(* CoDeSys 2.3.9.48 project: 20171120_WUR.pro *)
(* Version: 0.9 *)
(* Description: Project Distributie Automatisering *)
(* Libraries: Serial_Interface_01.lib 22.4.13 11:50:14, Util.lib 30.1.13 12:05:12, WagoLib787_01.lib 10.11.14 12:02:32, mod_com.lib 30.1.13 12:05:12, WagoConfigToolLIB.lib 30.1.13 12:05:12, PowerMeasurement_495_02.lib 25.8.17 14:41:17, SysLibTime.lib 30.1.13 12:05:12, WagoLibSHA1.lib 19.8.11 13:53:16, WagoLibMySQL_03.lib 23.7.14 08:13:36, SerComm.lib 30.1.13 12:05:12, SysLibSockets.lib 22.5.14 15:16:32, SysLibFile.lib 30.1.13 12:05:12, SysLibMem.lib 30.1.13 12:05:12, SysLibSem.lib 30.1.13 12:05:12, SysLibRtc.lib 30.1.13 12:05:12, WagoLibEthernet_01.lib 1.4.15 13:24:28, WAGOLIBNTP.lib 19.8.11 13:53:14, Modb_l05.lib 13.5.15 09:30:08, SysLibDir.lib 30.1.13 12:05:12, Standard.lib 20.5.14 07:13:26, Iecsfc.lib 30.1.13 12:05:12, SYSLIBCALLBACK.LIB 30.1.13 12:05:12, WagoLibModbus_IP_01.lib 12.2.16 10:20:24, Wago_MBCFG_ETHERNET_01.lib 1.4.15 13:24:28, Wago_MBCFG_COMMON_01.lib 1.4.15 13:24:28 *)

(* PLC configuration (modules and I/O channels)
0750-0430 8 DI 24 V DC 3.0ms [Type_1_8_Channels] node 1, in %IB264 out %QB280
  AT %IX132.0 [BOOLOnX_I] Ch_1 Digital input
  AT %IX132.1 [BOOLOnX_I] Ch_2 Digital input
  AT %IX132.2 [BOOLOnX_I] Ch_3 Digital input
  AT %IX132.3 [BOOLOnX_I] Ch_4 Digital input
  AT %IX132.4 [BOOLOnX_I] Ch_5 Digital input
  AT %IX132.5 [BOOLOnX_I] Ch_6 Digital input
  AT %IX132.6 [BOOLOnX_I] Ch_7 Digital input
  AT %IX132.7 [BOOLOnX_I] Ch_8 Digital input
0750-0430 8 DI 24 V DC 3.0ms [Type_1_8_Channels] node 2, in %IB264 out %QB280
  AT %IX132.8 [BOOLOnX_I] Ch_1 Digital input
  AT %IX132.9 [BOOLOnX_I] Ch_2 Digital input
  AT %IX132.10 [BOOLOnX_I] Ch_3 Digital input
  AT %IX132.11 [BOOLOnX_I] Ch_4 Digital input
  AT %IX132.12 [BOOLOnX_I] Ch_5 Digital input
  AT %IX132.13 [BOOLOnX_I] Ch_6 Digital input
  AT %IX132.14 [BOOLOnX_I] Ch_7 Digital input
  AT %IX132.15 [BOOLOnX_I] Ch_8 Digital input
0750-0430 8 DI 24 V DC 3.0ms [Type_1_8_Channels] node 3, in %IB265 out %QB280
  AT %IX133.0 [BOOLOnX_I] Ch_1 Digital input
  AT %IX133.1 [BOOLOnX_I] Ch_2 Digital input
  AT %IX133.2 [BOOLOnX_I] Ch_3 Digital input
  AT %IX133.3 [BOOLOnX_I] Ch_4 Digital input
  AT %IX133.4 [BOOLOnX_I] Ch_5 Digital input
  AT %IX133.5 [BOOLOnX_I] Ch_6 Digital input
  AT %IX133.6 [BOOLOnX_I] Ch_7 Digital input
  AT %IX133.7 [BOOLOnX_I] Ch_8 Digital input
0750-0430 8 DI 24 V DC 3.0ms [Type_1_8_Channels] node 4, in %IB266 out %QB280
  AT %IX133.8 [BOOLOnX_I] Ch_1 Digital input
  AT %IX133.9 [BOOLOnX_I] Ch_2 Digital input
  AT %IX133.10 [BOOLOnX_I] Ch_3 Digital input
  AT %IX133.11 [BOOLOnX_I] Ch_4 Digital input
  AT %IX133.12 [BOOLOnX_I] Ch_5 Digital input
  AT %IX133.13 [BOOLOnX_I] Ch_6 Digital input
  AT %IX133.14 [BOOLOnX_I] Ch_7 Digital input
  AT %IX133.15 [BOOLOnX_I] Ch_8 Digital input
0750-0430 8 DI 24 V DC 3.0ms [Type_1_8_Channels] node 5, in %IB267 out %QB280
  AT %IX134.0 [BOOLOnX_I] Ch_1 Digital input
  AT %IX134.1 [BOOLOnX_I] Ch_2 Digital input
  AT %IX134.2 [BOOLOnX_I] Ch_3 Digital input
  AT %IX134.3 [BOOLOnX_I] Ch_4 Digital input
  AT %IX134.4 [BOOLOnX_I] Ch_5 Digital input
  AT %IX134.5 [BOOLOnX_I] Ch_6 Digital input
  AT %IX134.6 [BOOLOnX_I] Ch_7 Digital input
  AT %IX134.7 [BOOLOnX_I] Ch_8 Digital input
0750-0530 8 DO 24 V DC 0.5A [Type_10_8_Channels] node 6, in %IB268 out %QB280
  AT %QX140.0 [BOOLOnX_Q] Ch_1 Digital output
  AT %QX140.1 [BOOLOnX_Q] Ch_2 Digital output
  AT %QX140.2 [BOOLOnX_Q] Ch_3 Digital output
  AT %QX140.3 [BOOLOnX_Q] Ch_4 Digital output
  AT %QX140.4 [BOOLOnX_Q] Ch_5 Digital output
  AT %QX140.5 [BOOLOnX_Q] Ch_6 Digital output
  AT %QX140.6 [BOOLOnX_Q] Ch_7 Digital output
  AT %QX140.7 [BOOLOnX_Q] Ch_8 Digital output
0750-0530 8 DO 24 V DC 0.5A [Type_10_8_Channels] node 7, in %IB269 out %QB280
  AT %QX140.8 [BOOLOnX_Q] Ch_1 Digital output
  AT %QX140.9 [BOOLOnX_Q] Ch_2 Digital output
  AT %QX140.10 [BOOLOnX_Q] Ch_3 Digital output
  AT %QX140.11 [BOOLOnX_Q] Ch_4 Digital output
  AT %QX140.12 [BOOLOnX_Q] Ch_5 Digital output
  AT %QX140.13 [BOOLOnX_Q] Ch_6 Digital output
  AT %QX140.14 [BOOLOnX_Q] Ch_7 Digital output
  AT %QX140.15 [BOOLOnX_Q] Ch_8 Digital output
0750-0530 8 DO 24 V DC 0.5A [Type_10_8_Channels] node 8, in %IB269 out %QB281
  AT %QX141.0 [BOOLOnX_Q] Ch_1 Digital output
  AT %QX141.1 [BOOLOnX_Q] Ch_2 Digital output
  AT %QX141.2 [BOOLOnX_Q] Ch_3 Digital output
  AT %QX141.3 [BOOLOnX_Q] Ch_4 Digital output
  AT %QX141.4 [BOOLOnX_Q] Ch_5 Digital output
  AT %QX141.5 [BOOLOnX_Q] Ch_6 Digital output
  AT %QX141.6 [BOOLOnX_Q] Ch_7 Digital output
  AT %QX141.7 [BOOLOnX_Q] Ch_8 Digital output
0750-0530 8 DO 24 V DC 0.5A [Type_10_8_Channels] node 9, in %IB269 out %QB282
  AT %QX141.8 [BOOLOnX_Q] Ch_1 Digital output
  AT %QX141.9 [BOOLOnX_Q] Ch_2 Digital output
  AT %QX141.10 [BOOLOnX_Q] Ch_3 Digital output
  AT %QX141.11 [BOOLOnX_Q] Ch_4 Digital output
  AT %QX141.12 [BOOLOnX_Q] Ch_5 Digital output
  AT %QX141.13 [BOOLOnX_Q] Ch_6 Digital output
  AT %QX141.14 [BOOLOnX_Q] Ch_7 Digital output
  AT %QX141.15 [BOOLOnX_Q] Ch_8 Digital output
0750-0555 4 AO 4-20mA [Type_14_4_Channels] node 10, in %IB240 out %QB256
  AT %QW0 [WORDOnW_Q] Ch_1 Analog output
  AT %QW1 [WORDOnW_Q] Ch_2 Analog output
  AT %QW2 [WORDOnW_Q] Ch_3 Analog output
  AT %QW3 [WORDOnW_Q] Ch_4 Analog output
0750-0559 4 AO 0-10V DC [Type_14_4_Channels] node 11, in %IB240 out %QB256
  AT %QW4 [WORDOnW_Q] Ch_1 Analog output
  AT %QW5 [WORDOnW_Q] Ch_2 Analog output
  AT %QW6 [WORDOnW_Q] Ch_3 Analog output
  AT %QW7 [WORDOnW_Q] Ch_4 Analog output
0750-0495/0000-0001 3-phase PoM690/ 5A [Type_58_1_Channels] node 12, in %IB240 out %QB264
  AT %IW0 [WORDOnW_I] Status Word
  AT %IW1 [WORDOnW_I] Status Word 1
  AT %IW2 [WORDOnW_I] Status Word 2
  AT %IW3 [WORDOnW_I] Status Word 3
  AT %ID2 [DWORDOnD_I] process value 1
  AT %ID3 [DWORDOnD_I] process value 2
  AT %ID4 [DWORDOnD_I] process value 3
  AT %ID5 [DWORDOnD_I] process value 4
  AT %QW8 [WORDOnW_Q] Control Word
  AT %QW9 [WORDOnW_Q] Control Word 1
  AT %QW10 [WORDOnW_Q] Control Word 2
  AT %QW11 [WORDOnW_Q] Control Word 3
0750-0495/0000-0001 3-phase PoM690/ 5A [Type_58_1_Channels] node 13, in %IB240 out %QB272
  AT %IW12 [WORDOnW_I] Status Word
  AT %IW13 [WORDOnW_I] Status Word 1
  AT %IW14 [WORDOnW_I] Status Word 2
  AT %IW15 [WORDOnW_I] Status Word 3
  AT %ID8 [DWORDOnD_I] process value 1
  AT %ID9 [DWORDOnD_I] process value 2
  AT %ID10 [DWORDOnD_I] process value 3
  AT %ID11 [DWORDOnD_I] process value 4
  AT %QW20 [WORDOnW_Q] Control Word
  AT %QW21 [WORDOnW_Q] Control Word 1
  AT %QW22 [WORDOnW_Q] Control Word 2
  AT %QW23 [WORDOnW_Q] Control Word 3
0750-0495/0000-0001 3-phase PoM690/ 5A [Type_58_1_Channels] node 14, in %IB264 out %QB296
  AT %IW24 [WORDOnW_I] Status Word
  AT %IW25 [WORDOnW_I] Status Word 1
  AT %IW26 [WORDOnW_I] Status Word 2
  AT %IW27 [WORDOnW_I] Status Word 3
  AT %ID14 [DWORDOnD_I] process value 1
  AT %ID15 [DWORDOnD_I] process value 2
  AT %ID16 [DWORDOnD_I] process value 3
  AT %ID17 [DWORDOnD_I] process value 4
  AT %QW32 [WORDOnW_Q] Control Word
  AT %QW33 [WORDOnW_Q] Control Word 1
  AT %QW34 [WORDOnW_Q] Control Word 2
  AT %QW35 [WORDOnW_Q] Control Word 3
0750-0495/0000-0001 3-phase PoM690/ 5A [Type_58_1_Channels] node 15, in %IB288 out %QB320
  AT %IW36 [WORDOnW_I] Status Word
  AT %IW37 [WORDOnW_I] Status Word 1
  AT %IW38 [WORDOnW_I] Status Word 2
  AT %IW39 [WORDOnW_I] Status Word 3
  AT %ID20 [DWORDOnD_I] process value 1
  AT %ID21 [DWORDOnD_I] process value 2
  AT %ID22 [DWORDOnD_I] process value 3
  AT %ID23 [DWORDOnD_I] process value 4
  AT %QW44 [WORDOnW_Q] Control Word
  AT %QW45 [WORDOnW_Q] Control Word 1
  AT %QW46 [WORDOnW_Q] Control Word 2
  AT %QW47 [WORDOnW_Q] Control Word 3
0750-0495/0000-0001 3-phase PoM690/ 5A [Type_58_1_Channels] node 16, in %IB312 out %QB344
  AT %IW48 [WORDOnW_I] Status Word
  AT %IW49 [WORDOnW_I] Status Word 1
  AT %IW50 [WORDOnW_I] Status Word 2
  AT %IW51 [WORDOnW_I] Status Word 3
  AT %ID26 [DWORDOnD_I] process value 1
  AT %ID27 [DWORDOnD_I] process value 2
  AT %ID28 [DWORDOnD_I] process value 3
  AT %ID29 [DWORDOnD_I] process value 4
  AT %QW56 [WORDOnW_Q] Control Word
  AT %QW57 [WORDOnW_Q] Control Word 1
  AT %QW58 [WORDOnW_Q] Control Word 2
  AT %QW59 [WORDOnW_Q] Control Word 3
0750-0495/0000-0001 3-phase PoM690/ 5A [Type_58_1_Channels] node 17, in %IB336 out %QB368
  AT %IW60 [WORDOnW_I] Status Word
  AT %IW61 [WORDOnW_I] Status Word 1
  AT %IW62 [WORDOnW_I] Status Word 2
  AT %IW63 [WORDOnW_I] Status Word 3
  AT %ID32 [DWORDOnD_I] process value 1
  AT %ID33 [DWORDOnD_I] process value 2
  AT %ID34 [DWORDOnD_I] process value 3
  AT %ID35 [DWORDOnD_I] process value 4
  AT %QW68 [WORDOnW_Q] Control Word
  AT %QW69 [WORDOnW_Q] Control Word 1
  AT %QW70 [WORDOnW_Q] Control Word 2
  AT %QW71 [WORDOnW_Q] Control Word 3
0750-0495/0000-0001 3-phase PoM690/ 5A [Type_58_1_Channels] node 18, in %IB360 out %QB392
  AT %IW72 [WORDOnW_I] Status Word
  AT %IW73 [WORDOnW_I] Status Word 1
  AT %IW74 [WORDOnW_I] Status Word 2
  AT %IW75 [WORDOnW_I] Status Word 3
  AT %ID38 [DWORDOnD_I] process value 1
  AT %ID39 [DWORDOnD_I] process value 2
  AT %ID40 [DWORDOnD_I] process value 3
  AT %ID41 [DWORDOnD_I] process value 4
  AT %QW80 [WORDOnW_Q] Control Word
  AT %QW81 [WORDOnW_Q] Control Word 1
  AT %QW82 [WORDOnW_Q] Control Word 2
  AT %QW83 [WORDOnW_Q] Control Word 3
0750-0495/0000-0001 3-phase PoM690/ 5A [Type_58_1_Channels] node 19, in %IB384 out %QB416
  AT %IW84 [WORDOnW_I] Status Word
  AT %IW85 [WORDOnW_I] Status Word 1
  AT %IW86 [WORDOnW_I] Status Word 2
  AT %IW87 [WORDOnW_I] Status Word 3
  AT %ID44 [DWORDOnD_I] process value 1
  AT %ID45 [DWORDOnD_I] process value 2
  AT %ID46 [DWORDOnD_I] process value 3
  AT %ID47 [DWORDOnD_I] process value 4
  AT %QW92 [WORDOnW_Q] Control Word
  AT %QW93 [WORDOnW_Q] Control Word 1
  AT %QW94 [WORDOnW_Q] Control Word 2
  AT %QW95 [WORDOnW_Q] Control Word 3
0750-0495/0000-0001 3-phase PoM690/ 5A [Type_58_1_Channels] node 20, in %IB408 out %QB440
  AT %IW96 [WORDOnW_I] Status Word
  AT %IW97 [WORDOnW_I] Status Word 1
  AT %IW98 [WORDOnW_I] Status Word 2
  AT %IW99 [WORDOnW_I] Status Word 3
  AT %ID50 [DWORDOnD_I] process value 1
  AT %ID51 [DWORDOnD_I] process value 2
  AT %ID52 [DWORDOnD_I] process value 3
  AT %ID53 [DWORDOnD_I] process value 4
  AT %QW104 [WORDOnW_Q] Control Word
  AT %QW105 [WORDOnW_Q] Control Word 1
  AT %QW106 [WORDOnW_Q] Control Word 2
  AT %QW107 [WORDOnW_Q] Control Word 3
0750-0495/0000-0001 3-phase PoM690/ 5A [Type_58_1_Channels] node 21, in %IB432 out %QB464
  AT %IW108 [WORDOnW_I] Status Word
  AT %IW109 [WORDOnW_I] Status Word 1
  AT %IW110 [WORDOnW_I] Status Word 2
  AT %IW111 [WORDOnW_I] Status Word 3
  AT %ID56 [DWORDOnD_I] process value 1
  AT %ID57 [DWORDOnD_I] process value 2
  AT %ID58 [DWORDOnD_I] process value 3
  AT %ID59 [DWORDOnD_I] process value 4
  AT %QW116 [WORDOnW_Q] Control Word
  AT %QW117 [WORDOnW_Q] Control Word 1
  AT %QW118 [WORDOnW_Q] Control Word 2
  AT %QW119 [WORDOnW_Q] Control Word 3
0750-0495/0000-0001 3-phase PoM690/ 5A [Type_58_1_Channels] node 22, in %IB456 out %QB488
  AT %IW120 [WORDOnW_I] Status Word
  AT %IW121 [WORDOnW_I] Status Word 1
  AT %IW122 [WORDOnW_I] Status Word 2
  AT %IW123 [WORDOnW_I] Status Word 3
  AT %ID62 [DWORDOnD_I] process value 1
  AT %ID63 [DWORDOnD_I] process value 2
  AT %ID64 [DWORDOnD_I] process value 3
  AT %ID65 [DWORDOnD_I] process value 4
  AT %QW128 [WORDOnW_Q] Control Word
  AT %QW129 [WORDOnW_Q] Control Word 1
  AT %QW130 [WORDOnW_Q] Control Word 2
  AT %QW131 [WORDOnW_Q] Control Word 3
Modbus variables [PFC200MODBUS] node 1, in %IB0 out %QB0 {PlcStopBehaviour = 1; FiledbusErrorBehaviour = 1; TcpOperation = 1; TcpPort = 502; TcpTimeout = 600; UdpOperation = 1; UdpPort = 502; RtuOperation = 0; NodeId = 1; ResponseTimeout = 5000; Interface = 0; Baud = 115200; StopBits = 1; Parity = 1; FlowCtrl = 0; PhysInterface = 0}
  REAL, Fieldbus output [MODBUS_REAL_OUT] node 0, in %IB0 out %QB0
    mb_var0 AT %QD500 [REALOnD_Q] TEST
Modbus-Master [MB_MASTER] node 2, in %IB0 out %QB0
*)

(* Task configuration *)
TASK Test (PRIORITY := 2, INTERVAL := T#500ms);
	Group1();
END_TASK
TASK WriteData (PRIORITY := 29); (* freewheeling *)
	Main_logger();
	SystemStateNames();
END_TASK
TASK GroupSwitching (PRIORITY := 4, INTERVAL := T#1000ms);
	run_group_switching();
END_TASK
TASK TestCHPSwitch (PRIORITY := 25, INTERVAL := T#100ms);
	CHP_switch_delay();
END_TASK
TASK LightControl (PRIORITY := 31); (* freewheeling *)
	error_lights();
END_TASK
TASK Measurements (PRIORITY := 1, INTERVAL := T#200ms);
	run_PQ();
	variables_to_system_array();
END_TASK
TASK Control (PRIORITY := 5, INTERVAL := T#100ms);
	CHP_Controller();
	SOC_to_Voltage_Out();
	Mixer_Controller1();
	Mixer_Controller2();
END_TASK
TASK MB_ETH_MASTER_TASK (PRIORITY := 3, INTERVAL := T#100ms);
	MBCFG_Janitza_UMG5090();
END_TASK
TASK SyncSwitch (PRIORITY := 2, INTERVAL := T#50ms);
	run_synchroniser_swtich();
END_TASK

(* Global variable list: Global_Variables *)
VAR_GLOBAL
(* testing purpose values *)
	x																:	 REAL:=2;

(* internally used variables *)
	r_Battery_Bus_Frequency									:	 REAL;
	r_Battery_Bus_Voltage										:	 REAL;
	r_Grid_Bus_Frequency										:	 REAL;
	r_Grid_Bus_Voltage											:	 REAL;


(* Array containing all the system parameters. Values are accessable through modbus tcp starting from register 12288. REAL uses two registers per variable *)
	arSystemState									AT %MW0	:	ARRAY[0.. iNumberSystemVar] OF REAL;
(*	arSystemStateNames										:	ARRAY[0.. iNumberSystemVar] OF STRING; (* names of registers used in mysql write *) *)

 (*Measurement values for cards*)
	arMeasurementsGroup1							:	ARRAY[1.. iNumberMeasurementVar] OF REAL;
	arMeasurementsGroup2							:	ARRAY[1.. iNumberMeasurementVar] OF REAL;
	arMeasurementsGroup3							:	ARRAY[1.. iNumberMeasurementVar] OF REAL;
	arMeasurementsGroup4							:	ARRAY[1.. iNumberMeasurementVar] OF REAL;
	arMeasurementsGroup5							:	ARRAY[1.. iNumberMeasurementVar] OF REAL;
	arMeasurementsGroup6							:	ARRAY[1.. iNumberMeasurementVar] OF REAL;
	arMeasurementsGroup7							:	ARRAY[1.. iNumberMeasurementVar] OF REAL;
	arMeasurementsGroup8							:	ARRAY[1.. iNumberMeasurementVar] OF REAL;
	arMeasurementsGroup9							:	ARRAY[1.. iNumberMeasurementVar] OF REAL;
	arMeasurementsGroupA							:	ARRAY[1.. iNumberMeasurementVar] OF REAL;
	arMeasurementsGroupB							:	ARRAY[1.. iNumberMeasurementVar] OF REAL;

 (*Measurement values for bus connector from janitza*)

	Bus_Connector_L1_P : REAL;
	Bus_Connector_L2_P : REAL;
	Bus_Connector_L3_P : REAL;
	Bus_Connector_L1_Q : REAL;
	Bus_Connector_L2_Q : REAL;
	Bus_Connector_L3_Q : REAL;
	Bus_Connector_L1_V : REAL;
	Bus_Connector_L2_V : REAL;
	Bus_Connector_L3_V : REAL;
	Bus_Connector_L1_I : REAL;
	Bus_Connector_L2_I : REAL;
	Bus_Connector_L3_I : REAL;
	Bus_Connector_L1_f : REAL;
	Bus_Connector_L2_f : REAL;
	Bus_Connector_L3_f : REAL;
	Bus_Connector_3F_CosPhi : REAL;
	Bus_Connector_3F_Field_Rotation: REAL;
	Bus_Connector_3F_radians: REAL;

(*  SYNCHRONISER SWITCH CONTROL *)

	Bus_Connector_3F_Sync_close_requested   			AT %QX141.2 : BOOL;
	Bus_Connector_3F_Sync_closed   						AT %IX133.12 : BOOL;
	Bus_Connector_3F_Sync_close_requested_panel    	AT %IX133.13 : BOOL;
	Bus_Connector_3F_Sync_denied_panel   				AT %IX133.14 : BOOL;
	Bus_Connector_3F_Sync_close_requested_modbus 					: BOOL;
	Bus_Connector_3F_Sync_denied_modbus				 				: BOOL;

(* CHP req	uest mode and control *)
	CHP_control_auto_bus_select_controlswitch 							: BOOL;
	CHP_control_Offgrid_request    							AT %QX141.4  : BOOL;
	CHP_control_internal_contacter_switch_state  			AT %IX134.3 : BOOL;
	CHP_relay_state_battery_bus   							AT %IX134.2  : BOOL;  (* INVERTED INPUTS *)
	CHP_relay_state_grid_bus   								AT %IX134.1  : BOOL;  (* INVERTED INPUTS *)

	CHP_new_state_battery_bus   							 : BOOL;
	CHP_new_state_grid_bus   								 : BOOL := TRUE;

(* not used any more, using input form group 1 relais
	CHP_control_grid_bus_select_controlswitch 							: BOOL;
	CHP_control_baterry_bus_select_controlswitch 						: BOOL;
	CHP_gridbus_switch_state												: BOOL; (*request from battery bus frequency *)
	CHP_batterybus_switch_state											: BOOL; (*request from battery bus frequency *)
*)

(* default auto swithcing parameters *)
	(* Frequencybased_bus_selecting_state							:  BOOL	:= TRUE; (* ?? not used ?? *) *)
	Group_control_Frequencybased_bus_selecting_state 			: BOOL:=TRUE;
	Switch_Gap_Time												:  INT		:= 10; (* seconds *)

	(* frequency based swithcing parameters *)
	Group_control_Frequencybased_parameters_initialized: BOOL :=FALSE;
	Group_control_min_time_above_switch_frequency : REAL := 20;
	Group_control_min_time_below_switch_frequency : REAL := 20;
	Group1_3F_Switch_frequency_to_batterybus : REAL := 49.5;
	Group1_3F_Switch_frequency_to_gridbus : REAL := 50;
	Group1_3F_min_time_between_switching : REAL:= 30;

	Group2_3F_Switch_frequency_to_batterybus : REAL := 49;
	Group2_3F_Switch_frequency_to_gridbus : REAL := 51;
	Group2_3F_min_time_between_switching : REAL := 10;

	Group3_3F_Switch_frequency_to_batterybus : REAL:= 49;
	Group3_3F_Switch_frequency_to_gridbus : REAL:= 51;
	Group3_3F_min_time_between_switching : REAL := 10;

	Group4_3F_Switch_frequency_to_batterybus : REAL:= 49;
	Group4_3F_Switch_frequency_to_gridbus : REAL:= 51;
	Group4_3F_min_time_between_switching : REAL := 10;

	Group5_3F_Switch_frequency_to_batterybus : REAL:= 49;
	Group5_3F_Switch_frequency_to_gridbus : REAL:= 51;
	Group5_3F_min_time_between_switching : REAL := 10;

	Group6_3F_Switch_frequency_to_batterybus : REAL:= 49;
	Group6_3F_Switch_frequency_to_gridbus : REAL:= 51;
	Group6_3F_min_time_between_switching : REAL := 10;

	Group7_3F_Switch_frequency_to_batterybus : REAL:= 49;
	Group7_3F_Switch_frequency_to_gridbus : REAL:= 51;
	Group7_3F_min_time_between_switching : REAL := 10;

	Group8_3F_Switch_frequency_to_batterybus : REAL:= 49;
	Group8_3F_Switch_frequency_to_gridbus : REAL:= 51;
	Group8_3F_min_time_between_switching : REAL := 10;

	Group9_3F_Switch_frequency_to_batterybus : REAL:= 49;
	Group9_3F_Switch_frequency_to_gridbus : REAL:= 51;
	Group9_3F_min_time_between_switching : REAL := 10;
(*
	Group4_gridbus_switch_automatic_request: BOOL :=TRUE;
	Group4_testbus_switch_automatic_request: BOOL :=FALSE;
	Group6_gridbus_switch_automatic_request: BOOL :=TRUE;
	Group6_testbus_switch_automatic_request: BOOL :=FALSE;
	Group9_gridbus_switch_automatic_request: BOOL :=TRUE;
	Group9_testbus_switch_automatic_request: BOOL :=FALSE;
	Groupx_gridbus_switch_automatic_request: BOOL :=TRUE;
	Groupx_testbus_switch_automatic_request: BOOL :=FALSE;

*)
(*
	Group1_Switch_frequency_to_batterybus						:  REAL	 := 52;
	Group1_Switch_frequency_to_gridbus							:  REAL	 := 48;
	Group1_min_time_above_switch_frequency					:  INT 		:= 10000; (*ms*)
	Group1_min_time_below_switch_frequency					:  INT 		:= 10000; (*ms*)
	Group1_min_time_between_switching							:  INT 		:= 10000; (*ms*)
	Group2_Switch_frequency_to_batterybus						:  REAL 	:= 52;
	Group2_Switch_frequency_to_gridbus							:  REAL 	:= 48;
	Group2_min_time_above_switch_frequency					:  INT 		:= 10000; (*ms*)
	Group2_min_time_below_switch_frequency					:  INT 		:= 10000; (*ms*)
	Group2_min_time_between_switching							:  INT 		:= 10000; (*ms*)
	Group3_Switch_frequency_to_batterybus						:  REAL 	:= 52;
	Group3_Switch_frequency_to_gridbus							:  REAL 	:= 48;
	Group3_min_time_above_switch_frequency					:  INT 		:= 10000; (*ms*)
	Group3_min_time_below_switch_frequency					:  INT 		:= 10000; (*ms*)
	Group3_min_time_between_switching							:  INT 		:= 10000; (*ms*)
	Group4_Switch_frequency_to_batterybus						:  REAL 	:= 52;
	Group4_Switch_frequency_to_gridbus							:  REAL 	:= 48;
	Group4_min_time_above_switch_frequency					:  INT 		:= 10000; (*ms*)
	Group4_min_time_below_switch_frequency					:  INT 		:= 10000; (*ms*)
	Group4_min_time_between_switching							:  INT 		:= 10000; (*ms*)
	Group5_Switch_frequency_to_batterybus						:  REAL 	:= 52;
	Group5_Switch_frequency_to_gridbus							:  REAL 	:= 48;
	Group5_min_time_above_switch_frequency					:  INT 		:= 10000; (*ms*)
	Group5_min_time_below_switch_frequency					:  INT 		:= 10000; (*ms*)
	Group5_min_time_between_switching							:  INT 		:= 10000; (*ms*)
	Group6_Switch_frequency_to_batterybus						:  REAL 	:= 52;
	Group6_Switch_frequency_to_gridbus							:  REAL 	:= 48;
	Group6_min_time_above_switch_frequency					:  INT 		:= 10000; (*ms*)
	Group6_min_time_below_switch_frequency					:  INT 		:= 10000; (*ms*)
	Group6_min_time_between_switching							:  INT 		:= 10000; (*ms*)
	Group7_Switch_frequency_to_batterybus						:  REAL 	:= 52;
	Group7_Switch_frequency_to_gridbus							:  REAL 	:= 48;
	Group7_min_time_above_switch_frequency					:  INT 		:= 10000; (*ms*)
	Group7_min_time_below_switch_frequency					:  INT 		:= 10000; (*ms*)
	Group7_min_time_between_switching							:  INT 		:= 10000; (*ms*)
	Group8_Switch_frequency_to_batterybus						:  REAL 	:= 52;
	Group8_Switch_frequency_to_gridbus							:  REAL 	:= 48;
	Group8_min_time_above_switch_frequency					:  INT 		:= 10000; (*ms*)
	Group8_min_time_below_switch_frequency					:  INT 		:= 10000; (*ms*)
	Group8_min_time_between_switching							:  INT 		:= 10000; (*ms*)
	Group9_Switch_frequency_to_batterybus						:  REAL 	:= 52;
	Group9_Switch_frequency_to_gridbus							:  REAL 	:= 48;
	Group9_min_time_above_switch_frequency					:  INT 		:= 10000; (*ms*)
	Group9_min_time_below_switch_frequency					:  INT 		:= 10000; (*ms*)
	Group9_min_time_between_switching							:  INT 		:= 10000; (*ms*)
*)

(* Analog Out Controller variables *)

	Mixer1_control_control_signal 							AT %QW4 : WORD;
	Mixer2_control_control_signal 							AT %QW6 : WORD; (*not in modbus! *)
	EV_control_control_signal   								AT %QW5 : WORD;
	other_control_control_signal   							AT %QW7 : WORD; (*not in modbus! *)

	CHP_control_Offgrid_Active_Power_control 			AT %QW0: WORD;	(*  *)
	mA_out2_control											AT %QW1: WORD;	(*not in modbus! *)
	mA_out3_control											AT %QW2: WORD;	(*not in modbus! *)
	mA_out4_control											AT %QW3: WORD;	(*not in modbus! *)

	Group1_3F_Auto_relay_control_battery_bus   	AT %QX140.1  : BOOL;
	Group1_3F_Auto_relay_control_grid_bus   		AT %QX140.0  : BOOL;
	Group1_3F_Selector_auto_bus_select    		AT %IX133.2 : BOOL;
	Group1_3F_relay_state_battery_bus   			AT %IX132.1  : BOOL;
	Group1_3F_relay_state_grid_bus   				AT %IX132.0  : BOOL;
	Group2_3F_Auto_relay_control_battery_bus   	AT %QX140.3  : BOOL;
	Group2_3F_Auto_relay_control_grid_bus   		AT %QX140.2  : BOOL;
	Group2_3F_Selector_auto_bus_select  			AT %IX133.3 : BOOL;
	Group2_3F_relay_state_battery_bus   			AT %IX132.3  : BOOL;
	Group2_3F_relay_state_grid_bus   				AT %IX132.2  : BOOL;
	Group3_3F_Auto_relay_control_battery_bus   	AT %QX140.5  : BOOL;
	Group3_3F_Auto_relay_control_grid_bus   		AT %QX140.4  : BOOL;
	Group3_3F_Selector_auto_bus_select   		AT %IX133.4 : BOOL;
	Group3_3F_relay_state_battery_bus   			AT %IX132.5  : BOOL;
	Group3_3F_relay_state_grid_bus   				AT %IX132.4  : BOOL;
	Group4_3F_Auto_relay_control_battery_bus    	AT %QX140.7  : BOOL;
	Group4_3F_Auto_relay_control_grid_bus    		AT %QX140.6  : BOOL;
	Group4_3F_Selector_auto_bus_select   		AT %IX133.5 : BOOL;
	Group4_3F_relay_state_battery_bus   			AT %IX132.7  : BOOL;
	Group4_3F_relay_state_grid_bus   				AT %IX132.6  : BOOL;
	Group5_3F_Auto_relay_control_battery_bus   	AT %QX140.9  : BOOL;
	Group5_3F_Auto_relay_control_grid_bus   		AT %QX140.8  : BOOL;
	Group5_3F_Selector_auto_bus_select   		AT %IX133.6 : BOOL;
	Group5_3F_relay_state_battery_bus   			AT %IX132.9  : BOOL;
	Group5_3F_relay_state_grid_bus   				AT %IX132.8  : BOOL;
	Group6_3F_Auto_relay_control_battery_bus   	AT %QX140.11  : BOOL;
	Group6_3F_Auto_relay_control_grid_bus   		AT %QX140.10  : BOOL;
	Group6_3F_Selector_auto_bus_select   		AT %IX133.7 : BOOL;
	Group6_3F_relay_state_battery_bus   			AT %IX132.11  : BOOL;
	Group6_3F_relay_state_grid_bus   				AT %IX132.10  : BOOL;
	Group7_3F_Auto_relay_control_battery_bus   	AT %QX140.13  : BOOL;
	Group7_3F_Auto_relay_control_grid_bus   		AT %QX140.12  : BOOL;
	Group7_3F_Selector_auto_bus_select   		AT %IX133.8 : BOOL;
	Group7_3F_relay_state_battery_bus   			AT %IX132.13  : BOOL;
	Group7_3F_relay_state_grid_bus   				AT %IX132.12  : BOOL;
	Group8_3F_Auto_relay_control_battery_bus   	AT %QX140.15  : BOOL;
	Group8_3F_Auto_relay_control_grid_bus   		AT %QX140.14  : BOOL;
	Group8_3F_Selector_auto_bus_select   		AT %IX133.9 : BOOL;
	Group8_3F_relay_state_battery_bus   			AT %IX132.15  : BOOL;
	Group8_3F_relay_state_grid_bus   				AT %IX132.14  : BOOL;
	Group9_3F_Auto_relay_control_battery_bus   	AT %QX141.1  : BOOL;
	Group9_3F_Auto_relay_control_grid_bus   		AT %QX141.0  : BOOL;
	Group9_3F_Selector_auto_bus_select   		AT %IX133.10 : BOOL;
	Group9_3F_relay_state_battery_bus   			AT %IX133.1  : BOOL;
	Group9_3F_relay_state_grid_bus   				AT %IX133.0  : BOOL;

(* Controm panel LEDs *)
	Control_panel_status_operational_led    		AT %QX141.11  : BOOL;
	Control_panel_status_warning_led   			AT %QX141.12  : BOOL;
	Control_panel_status_error_led   				AT %QX141.13  : BOOL;

(* TheBattery setting *)
	TheBattery_SOC_real : REAL;
	TheBattery_SOC_simulated : REAL;
	TheBattery_bool_use_PLC_SOC : REAL;
	TheBattery_SOC_PLC_SOC_setpoint : REAL;

(* TEST SETTINGS CHP SWICHT HANDLER *)
      (* EV_control_control_signal3 :REAL;
	other_control_control_signal3:REAL;*)
	other_control_control_signal2 : REAL; (*not in modbus! *)
	Grid_IN: BOOL;
	BAT_out: BOOL;
	Grid_OUT: BOOL;
	BAT_IN: BOOL;

	time_below_switch_frequency: INT;
	time_above_switch_frequency: INT;
END_VAR

VAR_GLOBAL CONSTANT

(* System array length *)
	iNumberSystemVar			:	INT := 350;
(* measurement array length *)
	iNumberMeasurementVar		:	INT := 18;
	iNumberMeasurementGroups	:	 INT:= 11;

(* MySQL *)
	gcMySql_iSqlLength			:	 INT := 370; 		(* Defines the size in byte of an array element of "asSqlStatement", used by function blocks "MySql_ExecSql" and "MySql_Query"
															to provide an SQL statement as "ARRAY [0..UpperBound] OF STRING(Size)".*)
	raw_SQL_STR_LENGTH		:	 INT := 350;

	gc_MaxBufferSize 	       :INT := 5; (*number of items to hold in memory*)
	gv_iBuffCounter			:INT := 0; (* counter for  buffer*)
	gv_iBuffPointer			:INT := 0; (* pointer  for  buffer*)
	gv_Buffer					:ARRAY[0..gc_MaxBufferSize] OF ARRAY[0.. iNumberSystemVar] OF REAL; (*In memory buffer of failed message attempts*)
	gc_LogInterval			:TIME := t#1s;
	gc_variables_to_write	:INT:=2;

	gc_sHost : STRING := '192.168.1.9';  (*'application.dyndns.info';*)
	gc_uiPort : UINT := 3306;
	gc_sUser : STRING := 'acrres'; (*'Acrres_write';*)
	gc_sPwd : STRING := 'Acrres123';(*'Acrres123';*)
	gc_sDB : STRING := 'Acrres';   	(* Optional - Name of database instance to connect to *)
	gc_sTable:STRING := 'Switch_container' ;

(* Read / write CSV-files *)
	iMaxParams			:	INT:=8;(* Number of Parameters per File *)
	gc_ParameterCount	:	INT:=1;(* Number of Values per Parameter *)
	gc_RawDataSize		:	UINT:=500; (* Raw data size for reading in file ASCII *)
	gcRowExcel			:	INT:=1;


END_VAR

VAR_GLOBAL PERSISTENT RETAIN
(* also set in hardware itself, seems like this is not really used in de measurement code, even though it given as input/setup... should be checked with current clams*)
	CurrentRatioPQ1						:	WORD := 300;		(* Current transformer ratio, eg 5 A / 300 A >>> 1:60, which was set in the hardware..*)
	CurrentRatioPQ2						:	WORD := 200;		(* Current transformer ratio, eg 5 A / 200 A >>> 1:40, which was set in the hardware..*)
	CurrentRatioPQ3						:	WORD := 200;		(* Current transformer ratio, eg 5 A / 200 A >>> 1:40, which was set in the hardware..*)
	CurrentRatioPQ4						:	WORD := 100;		(* Current transformer ratio, eg 5 A / 100 A >>> 1:20, which was set in the hardware..*)
	CurrentRatioPQ5						:	WORD := 100;		(* Current transformer ratio, eg 5 A / 100 A >>> 1:20, which was set in the hardware..*)
	CurrentRatioPQ6						:	WORD := 100;		(* Current transformer ratio, eg 5 A / 100 A >>> 1:20, which was set in the hardware..*)
	CurrentRatioPQ7						:	WORD := 100;		(* Current transformer ratio, eg 5 A / 100 A >>> 1:20, which was set in the hardware..*)
	CurrentRatioPQ8						:	WORD := 100;		(* Current transformer ratio, eg 5 A / 100 A >>> 1:20, which was set in the hardware..*)
	CurrentRatioPQ9						:	WORD := 100;		(* Current transformer ratio, eg 5 A / 100 A >>> 1:20, which was set in the hardware..*)
	CurrentRatioPQA						:	WORD := 400;		(* Current transformer ratio, eg 5 A / 400 A >>> 1:80, which was set in the hardware..*)
	CurrentRatioPQB						:	WORD := 400;		(* Current transformer ratio, eg 5 A / 400 A >>> 1:80, which was set in the hardware..*)

END_VAR

(* Data type *)
TYPE typCSV :
STRUCT
	sDescription	:STRING;
	Parameter		:ARRAY[1..gc_ParameterCount] OF STRING;
END_STRUCT
END_TYPE

(* POU 04. Frequency based Bus Select/Group1, FBD *)
PROGRAM Group1
VAR
	Switch: Auto_switch_new;
	temp: BOOL;
END_VAR
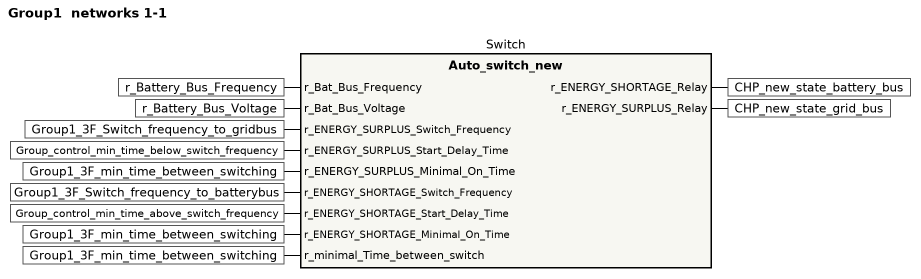
_FBD_ (* Function Block Diagram *)
NETWORK 1
	Switch:Auto_switch_new(r_Bat_Bus_Frequency: r_Battery_Bus_Frequency, r_Bat_Bus_Voltage: r_Battery_Bus_Voltage, r_ENERGY_SURPLUS_Switch_Frequency: Group1_3F_Switch_frequency_to_gridbus, r_ENERGY_SURPLUS_Start_Delay_Time: Group_control_min_time_below_switch_frequency, r_ENERGY_SURPLUS_Minimal_On_Time: Group1_3F_min_time_between_switching, r_ENERGY_SHORTAGE_Switch_Frequency: Group1_3F_Switch_frequency_to_batterybus, r_ENERGY_SHORTAGE_Start_Delay_Time: Group_control_min_time_above_switch_frequency, r_ENERGY_SHORTAGE_Minimal_On_Time: Group1_3F_min_time_between_switching, r_minimal_Time_between_switch: Group1_3F_min_time_between_switching, r_ENERGY_SURPLUS_Relay => CHP_new_state_grid_bus) => CHP_new_state_battery_bus
_END_FBD_
(* the same logic as Structured Text *)
(* Network 1 *)
Switch(r_Bat_Bus_Frequency := r_Battery_Bus_Frequency, r_Bat_Bus_Voltage := r_Battery_Bus_Voltage, r_ENERGY_SURPLUS_Switch_Frequency := Group1_3F_Switch_frequency_to_gridbus, r_ENERGY_SURPLUS_Start_Delay_Time := Group_control_min_time_below_switch_frequency, r_ENERGY_SURPLUS_Minimal_On_Time := Group1_3F_min_time_between_switching, r_ENERGY_SHORTAGE_Switch_Frequency := Group1_3F_Switch_frequency_to_batterybus, r_ENERGY_SHORTAGE_Start_Delay_Time := Group_control_min_time_above_switch_frequency, r_ENERGY_SHORTAGE_Minimal_On_Time := Group1_3F_min_time_between_switching, r_minimal_Time_between_switch := Group1_3F_min_time_between_switching);
CHP_new_state_grid_bus := Switch.r_ENERGY_SURPLUS_Relay;
CHP_new_state_battery_bus := Switch.r_ENERGY_SHORTAGE_Relay;
END_PROGRAM

(* POU 04. Frequency based Bus Select/Auto_switch_new, ST *)
FUNCTION_BLOCK Auto_switch_new
VAR_INPUT

	r_Bat_Bus_Frequency							:	REAL;
	r_Bat_Bus_Voltage								:	REAL;
	r_ENERGY_SURPLUS_Switch_Frequency		:	REAL := 51;
	r_ENERGY_SURPLUS_Start_Delay_Time		:	REAL := 5;
	r_ENERGY_SURPLUS_Minimal_On_Time		:	REAL;			(*not used*)
	r_ENERGY_SHORTAGE_Switch_Frequency	:	REAL := 49;
	r_ENERGY_SHORTAGE_Start_Delay_Time		:	REAL := 5;
	r_ENERGY_SHORTAGE_Minimal_On_Time	:	REAL; 			(*not used*)
	r_minimal_Time_between_switch				: 	REAL := 10;	(* Time between on and off grid relay switching (dead bus gap) *)

END_VAR
VAR_OUTPUT

	r_ENERGY_SHORTAGE_Relay								:	BOOL := TRUE;
	r_ENERGY_SURPLUS_Relay								:	BOOL;

END_VAR
VAR
	(*r_Test_Frequency							:	REAL:=50;*)
	r_Bat_Bus_Min_Voltage 							: 	REAL :=200;
	r_Checked_Grid_Bus_Start_Frequency			:	REAL;
	r_Checked_Bat_Bus_Start_Frequency			:	REAL;
(*
	t_Grid_Bus_Start_Delay_Timer					:	TON;
	t_Bat_Bus_Start_Delay_Timer					:	TON;
	t_minimal_switch_time_Delay_Timer			:	TON;
*)
	time_since_switch: INT := 0;
	min_time_below_safe_voltage: INT := 4;
	time_below_safe_voltage: INT := 0;
	time_below_switch_frequency: INT := 0;
	time_above_switch_frequency: INT := 0;
	run_time: INT := 0;
	current_state: REAL := 0;
END_VAR
(*
this script shuold run every second and 

------ Cases 1 - SAFETY ------
1) bat voltage  below 200 	> swtich to gridbus
------ Cases 2 - NO PENDEL ------
2) just switched (wait for r_Switch_Gap_Time)

------ Cases 3 - LOW FREQUENCY = ENERGY SHORTAGE ------
3a) bat frequency  > r_ENERGY_SHORTAGE_Switch_Frequency => "reset "ENERGY SHORTAGE counter"
3b) bat frequency  < r_ENERGY_SHORTAGE_Switch_Frequency => "increase "ENERGY SHORTAGE counter"
3c) "to grid counter" > r_Grid_Bus_Start_Delay_Time => switch of testbus, switch on gridbus relais 

------ Cases 4 - HIGH FREQUENCY = ENERGY SURPLUS ------
4a) bat frequency > r_ENERGY_SURPLUS_Switch_Frequency => "increase "to grid counter"
4b) bat frequency  < r_ENERGY_SURPLUS_Switch_Frequency => "reset "to bat counter"
4c) "to bat counter" > r_Grid_Bus_Start_Delay_Time => switch of gridbus, switch on testbus relais 
*)
run_time := run_time +1;
IF r_Bat_Bus_Voltage < r_Bat_Bus_Min_Voltage THEN
	current_state:=1;
	(* case 1 (safety, switching to gridbus after 2 seconds) *)
	IF time_below_safe_voltage < min_time_below_safe_voltage THEN
		time_below_safe_voltage := time_below_safe_voltage + 1;
		current_state:=1.2;
	ELSE
		r_ENERGY_SURPLUS_Relay := FALSE;
		r_ENERGY_SHORTAGE_Relay := TRUE;
		time_since_switch := 0;
		current_state:=1.4;
	END_IF

ELSE
	current_state:=2;
	IF time_since_switch < REAL_TO_INT(r_minimal_Time_between_switch) THEN
	(* case 2 (already switched recently) *)
	time_below_safe_voltage := 0;
	time_since_switch := time_since_switch + 1;
	current_state:=2.2;
	END_IF
END_IF

IF time_since_switch >= REAL_TO_INT(r_minimal_Time_between_switch) THEN
	(* CASE 3 *)
	(* 3a+b *)
	current_state:=3;
	(*IF r_Bat_Bus_Frequency < r_ENERGY_SHORTAGE_Switch_Frequency THEN*) (*MAX(r_Bat_Bus_Frequency, r_ENERGY_SHORTAGE_Switch_Frequency) = r_ENERGY_SHORTAGE_Switch_Frequency*)
	IF r_Bat_Bus_Frequency < r_ENERGY_SHORTAGE_Switch_Frequency THEN
		time_below_switch_frequency := time_below_switch_frequency + 1;
		current_state:=3.2;
	ELSE
		time_below_switch_frequency := 0;
		current_state:=3.4;
	END_IF

	(* 3C time_below_switch_frequency passed >> switching *)
	IF r_ENERGY_SURPLUS_Relay THEN
		IF time_below_switch_frequency > REAL_TO_INT(r_ENERGY_SHORTAGE_Start_Delay_Time) THEN
			current_state:=3.6;
			r_ENERGY_SURPLUS_Relay := FALSE;
			r_ENERGY_SHORTAGE_Relay := TRUE;
			time_since_switch := 0;
		END_IF
	END_IF

	(* CASE 4 *)
	(* 4a+b *)
	IF r_Bat_Bus_Frequency > r_ENERGY_SURPLUS_Switch_Frequency THEN
		time_above_switch_frequency := time_above_switch_frequency + 1;
		(*current_state:=4.2;*)
	ELSE
		time_above_switch_frequency := 0;
		(*current_state:=4.4;*)
	END_IF

	(* 4C time_above_switch_frequency passed >> switching*)
	IF r_ENERGY_SHORTAGE_Relay THEN
		IF time_above_switch_frequency > REAL_TO_INT(r_ENERGY_SURPLUS_Start_Delay_Time) THEN
			r_ENERGY_SHORTAGE_Relay := FALSE;
			r_ENERGY_SURPLUS_Relay := TRUE;
			time_since_switch := 0;
			(*current_state:=4.6;*)
		END_IF
	END_IF
END_IF
END_FUNCTION_BLOCK

(* POU 04. Frequency based Bus Select/temp, ST *)
PROGRAM temp
VAR
	b_DI_Group_AskedState_Grid					:	BOOL; (* NOT jet available !!!!!!!!!!! *)
	b_DI_Group_AskedState_Battery				:	BOOL; (* NOT jet available !!!!!!!!!!! *)
	b_DI_Group_AskedState_Auto					:	BOOL;
	b_DI_CHP_Sync_Contactor						:	BOOL;
	b_batbus_switch_state							:	BOOL;
	b_gridbus_switch_state							:	BOOL;
END_VAR
(* what happens when no automated switching is performed? REQUESTED STATE IS DETERMINED BY RELAIS STATE *)
	IF b_DI_Group_AskedState_Grid THEN
		b_Wanted_state_To_CHP := FALSE;

		(*IF r_BAT_BUS_Grid_Relay THEN*)
			IF  b_DI_CHP_Sync_Contactor = FALSE THEN
				b_Grid_Relay := FALSE;
				b_Bat_Relay := TRUE;
			END_IF
		(*END_IF*)
	ELSE IF b_DI_Group_AskedState_Battery THEN
		(*r_Wanted_state_To_CHP := TRUE;*)

		(*IF r_On_Grid_Relay THEN*)
			IF  b_DI_CHP_Sync_Contactor = FALSE THEN
					b_Bat_Relay := TRUE;
					b_Grid_Relay := FALSE;
			END_IF
		(*END_IF*)
	ELSE
		(* performe swithcing (only when CHP is disconnected) *)
		IF b_Bat_Relay THEN
				IF  b_DI_CHP_Sync_Contactor = FALSE THEN
						b_Bat_Relay := FALSE;
						b_Grid_Relay := TRUE;
				END_IF
		END_IF
		IF b_Grid_Relay THEN
				IF  b_DI_CHP_Sync_Contactor = FALSE THEN
						b_Bat_Relay := TRUE;
						b_Grid_Relay := FALSE;
				END_IF
		END_IF
END_IF
END_IF


(* ____________________________ OLD ___________________________ *)
Group1_gridbus_switch_state := r_Grid_Relay;
Group1_batterybus_switch_state := r_Bat_Relay;

(* parameters *)
Group_control_Frequencybased_bus_selecting_state
r_DI_Group_AskedState_Grid := Group1_autoswitch_state;
r_DI_CHP_Sync_Contactor: = CHP_control_internal_contacter_switch_state;
Group1_autoswitch_state

CHP_gridbus_switch_state 		(* request based on frequency *)
CHP_batterybus_switch_state  	(* request based on frequency *)
END_PROGRAM

(* POU 06. Mysql Write/Main_logger, ST *)
PROGRAM Main_logger
VAR


	xDoIt : BOOL;
	wState : WORD; (* Statemachine*)
	oMySql : MySql_Context; (* Used like Structure for keeping login and status information - Do not call it with in your program *)

	hasBufferedItems :  BOOL; (*Flag indicating the status of the buffer *)
	TONInst : TON; (* Sleep timer  *)

	(* Functionblock to contact MySql server *)
	oMySqlLogin : MySql_Login;

	xConnect : BOOL;
	diErrorLogin : DINT;
	sStatusLogin : STRING(500);
	xConnected : BOOL;

	(* Functionblock to process SQL statements who do not return result sets *)
	oMySqlExec1 : MySql_Execute;
	asSqlStatement1 : ARRAY [0..gcMySql_iSqlUpperBound] OF STRING(gcMySql_iSqlLength);
	xExec1 : BOOL;
	diErrorExec1 : DINT;
	sStatusExec1 : STRING(700);

	(*TODO clean this up these might be unnecassar delete if not used *)
	(* Functionblock to process SQL statements who return result sets *)
	oMySqlQuery1 : MySql_Query;
	asSqlQuery1 : ARRAY [0..gcMySql_iSqlUpperBound] OF STRING(gcMySql_iSqlLength);
	xQuery1 : BOOL;
	diErrorQuery1 : DINT;
	sStatusQuery1 : STRING(500);
	stQueryResult1 : MySql_ResultSet;

	(* Functionblock to disconnect MySql server *)
	oMySqlLogout : MySql_Logout;
	xDisconnect : BOOL;
	diErrorLogout : DINT;
	sStatusLogout : STRING(500);

	(* Helpers *)
	iHelp : INT;
	i : INT;
	END_: BOOL;
	strTempSQLStatement: STRING(raw_SQL_STR_LENGTH);


	(* debug variables *)
	iCountExecFailed: INT;
	xDolt: BOOL;

	stSystime: REAL;
END_VAR
(* Call function block "MySql_Login" every cycle to monitor connection status *)

oMySqlLogin(sHost:= gc_sHost,
			uiPort:= gc_uiPort,
			sUsername:= gc_sUser,
			sPassword:= gc_sPwd,
			sDatabase:=gc_sDB,
			oMySql:= oMySql,
			xStart:= xConnect,
			diError=> diErrorLogin,
			sStatus=> sStatusLogin,
			xConnected=> xConnected);

(*Get system time *)
(*
stSystime := Get_Time();
*)

CASE wState OF
0:

	xConnect := TRUE;
	wState := 10;

10:
	IF xConnected THEN

		xConnect := FALSE;
		IF TRUE  THEN  (*  Check that our power measurment model  is ready *)
			wState := 20; (* Proceede to execute SQL*)
		ELSE
			(* this is a different error state *)
			wState:= 45; (* wait and go to holding pattern for power measurement sensor to be ready*)
		END_IF
	ELSE
		wstate:=0;
	END_IF

20: (* prepare sql statement *)
	asSqlStatement1  := SQLStatement(    s_Table:= gc_sTable,
											);
	xExec1 := TRUE; (* Execute SQL-Insert-Statement *)
	wState :=25;

25:
	oMySqlExec1(asSqlCommand:=asSqlStatement1,
					oMySql:=oMySql,
					xStart:=xExec1,
					diError=> diErrorExec1,
					sStatus=>sStatusExec1);

	IF NOT  xExec1 THEN
		(* success *)
		xDisconnect := TRUE;
		wState := 50;  (*finished go and disconnect or start again *);

	ELSE

		(* Failed *)
		iCountExecFailed := iCountExecFailed +1; (* TODO count number of failures and fire an alarm *)
		wState:=50;

	END_IF


45: (* Wait here to debug convert problem *)
	(* buffer current value into memory *)
	(*
	IF gv_iBuffCounter < gc_MaxBufferSize THEN
		gv_Buffer[gv_iBuffCounter] := arCurrDataPoint; (* add data point to our buffer *)
		gv_iBuffCounter := gv_iBuffCounter + 1; (* incremenr buffer counter *)
		hasBufferedItems := TRUE; (*Flag indicating the status of the buffer *)
	END_IF
	*)
	wState := 60; (*move onto sleep*)

(*sleep X amount of time and continue*)


50: (* Disconnect from database *)
	oMySqlLogout(oMySql:= oMySql,
				 xStart:= xDisconnect,
				 diError=> diErrorLogout,
				 sStatus=> sStatusLogout);
	IF NOT xDisconnect THEN
		xDoIt := FALSE;
		wState := 60;(*move onto sleep*)
	END_IF

60:
	(*sleep X amount of time and continue*)
	TONInst( IN:= TRUE, PT := gc_LogInterval);

	IF TONInst.Q THEN
			wState := 0;
	(* ELSE do nothing just wait*)
	END_IF

END_CASE
END_PROGRAM

(* POU 06. Mysql Write/SQLStatement, ST *)
FUNCTION SQLStatement : ARRAY [0..gcMySql_iSqlUpperBound] OF STRING(gcMySql_iSqlLength)
VAR_INPUT

	s_Table 						: 	STRING;

END_VAR

VAR

	i	:	 INT;
	j	:	 INT;

	stNameArrayString	:	STRING;


END_VAR
SystemStateNames();

SQLStatement[0] := 'INSERT INTO `Acrres`.`';
SQLStatement[1] := s_Table;
SQLStatement[2] :=  '` (`datetime';
(*gc_variables_to_write : = iNumberSystemVar;*)
j:=3;
FOR i := 1 TO gc_variables_to_write DO

	SQLStatement[j] := CONCAT('`,`',arSystemStateNames[i]);
	j:= j+1;

END_FOR

SQLStatement[j] := CONCAT('`) VALUES (NOW(',')'); (*from_unixtime(',REAL_TO_STRING(arSystemState[0]));*)
j:=j+1;
(* SQLStatement[j] := ')';
j:=j+1;
*)

FOR i := 1 TO gc_variables_to_write DO
	SQLStatement[j] :=  CONCAT(',',REAL_TO_STRING(arSystemState[i]));
	j:=j+1;
END_FOR

SQLStatement[j] :=  ');';
END_FUNCTION

(* POU 06. Mysql Write/SystemStateNames, ST *)
PROGRAM SystemStateNames
VAR
END_VAR
(* update this list  via https://docs.google.com/spreadsheets/d/1TR7oXGZyEmNnGigmreKdtnpXsz8mxFcoB4b4beNITCA/edit#gid=0 *)
	arSystemStateNames[1] :='GroupA_L1_P';
	arSystemStateNames[2] :='GroupA_L2_P';
	arSystemStateNames[3] :='GroupA_L3_P';
	arSystemStateNames[4] :='GroupA_L1_Q';
	arSystemStateNames[5] :='GroupA_L2_Q';
	arSystemStateNames[6] :='GroupA_L3_Q';
	arSystemStateNames[7] :='GroupA_L1_V';
	arSystemStateNames[8] :='GroupA_L2_V';
	arSystemStateNames[9] :='GroupA_L3_V';
	arSystemStateNames[10] :='GroupA_L1_I';
	arSystemStateNames[11] :='GroupA_L2_I';
	arSystemStateNames[12] :='GroupA_L3_I';
	arSystemStateNames[13] :='GroupA_L1_f';
	arSystemStateNames[14] :='GroupA_L2_f';
	arSystemStateNames[15] :='GroupA_L3_f';
	arSystemStateNames[16] :='GroupA_3F_E';
	arSystemStateNames[17] :='GroupA_3F_Field_Rotation';
	arSystemStateNames[18] :='GroupA_3F_E_Reactive';
	arSystemStateNames[19] :='GroupB_L1_P';
	arSystemStateNames[20] :='GroupB_L2_P';
	arSystemStateNames[21] :='GroupB_L3_P';
	arSystemStateNames[22] :='GroupB_L1_Q';
	arSystemStateNames[23] :='GroupB_L2_Q';
	arSystemStateNames[24] :='GroupB_L3_Q';
	arSystemStateNames[25] :='GroupB_L1_V';
	arSystemStateNames[26] :='GroupB_L2_V';
	arSystemStateNames[27] :='GroupB_L3_V';
	arSystemStateNames[28] :='GroupB_L1_I';
	arSystemStateNames[29] :='GroupB_L2_I';
	arSystemStateNames[30] :='GroupB_L3_I';
	arSystemStateNames[31] :='GroupB_L1_f';
	arSystemStateNames[32] :='GroupB_L2_f';
	arSystemStateNames[33] :='GroupB_L3_f';
	arSystemStateNames[34] :='GroupB_3F_E';
	arSystemStateNames[35] :='GroupB_3F_Field_Rotation';
	arSystemStateNames[36] :='GroupB_3F_E_Reactive';
	arSystemStateNames[37] :='Group1_L1_P';
	arSystemStateNames[38] :='Group1_L2_P';
	arSystemStateNames[39] :='Group1_L3_P';
	arSystemStateNames[40] :='Group1_L1_Q';
	arSystemStateNames[41] :='Group1_L2_Q';
	arSystemStateNames[42] :='Group1_L3_Q';
	arSystemStateNames[43] :='Group1_L1_V';
	arSystemStateNames[44] :='Group1_L2_V';
	arSystemStateNames[45] :='Group1_L3_V';
	arSystemStateNames[46] :='Group1_L1_I';
	arSystemStateNames[47] :='Group1_L2_I';
	arSystemStateNames[48] :='Group1_L3_I';
	arSystemStateNames[49] :='Group1_L1_f';
	arSystemStateNames[50] :='Group1_L2_f';
	arSystemStateNames[51] :='Group1_L3_f';
	arSystemStateNames[52] :='Group1_3F_E';
	arSystemStateNames[53] :='Group1_3F_Field_Rotation';
	arSystemStateNames[54] :='Group1_3F_E_Reactive';
	arSystemStateNames[55] :='Group2_L1_P';
	arSystemStateNames[56] :='Group2_L2_P';
	arSystemStateNames[57] :='Group2_L3_P';
	arSystemStateNames[58] :='Group2_L1_Q';
	arSystemStateNames[59] :='Group2_L2_Q';
	arSystemStateNames[60] :='Group2_L3_Q';
	arSystemStateNames[61] :='Group2_L1_V';
	arSystemStateNames[62] :='Group2_L2_V';
	arSystemStateNames[63] :='Group2_L3_V';
	arSystemStateNames[64] :='Group2_L1_I';
	arSystemStateNames[65] :='Group2_L2_I';
	arSystemStateNames[66] :='Group2_L3_I';
	arSystemStateNames[67] :='Group2_L1_f';
	arSystemStateNames[68] :='Group2_L2_f';
	arSystemStateNames[69] :='Group2_L3_f';
	arSystemStateNames[70] :='Group2_3F_E';
	arSystemStateNames[71] :='Group2_3F_Field_Rotation';
	arSystemStateNames[72] :='Group2_3F_E_Reactive';
	arSystemStateNames[73] :='Group3_L1_P';
	arSystemStateNames[74] :='Group3_L2_P';
	arSystemStateNames[75] :='Group3_L3_P';
	arSystemStateNames[76] :='Group3_L1_Q';
	arSystemStateNames[77] :='Group3_L2_Q';
	arSystemStateNames[78] :='Group3_L3_Q';
	arSystemStateNames[79] :='Group3_L1_V';
	arSystemStateNames[80] :='Group3_L2_V';
	arSystemStateNames[81] :='Group3_L3_V';
	arSystemStateNames[82] :='Group3_L1_I';
	arSystemStateNames[83] :='Group3_L2_I';
	arSystemStateNames[84] :='Group3_L3_I';
	arSystemStateNames[85] :='Group3_L1_f';
	arSystemStateNames[86] :='Group3_L2_f';
	arSystemStateNames[87] :='Group3_L3_f';
	arSystemStateNames[88] :='Group3_3F_E';
	arSystemStateNames[89] :='Group3_3F_Field_Rotation';
	arSystemStateNames[90] :='Group3_3F_E_Reactive';
	arSystemStateNames[91] :='Group4_L1_P';
	arSystemStateNames[92] :='Group4_L2_P';
	arSystemStateNames[93] :='Group4_L3_P';
	arSystemStateNames[94] :='Group4_L1_Q';
	arSystemStateNames[95] :='Group4_L2_Q';
	arSystemStateNames[96] :='Group4_L3_Q';
	arSystemStateNames[97] :='Group4_L1_V';
	arSystemStateNames[98] :='Group4_L2_V';
	arSystemStateNames[99] :='Group4_L3_V';
	arSystemStateNames[100] :='Group4_L1_I';
	arSystemStateNames[101] :='Group4_L2_I';
	arSystemStateNames[102] :='Group4_L3_I';
	arSystemStateNames[103] :='Group4_L1_f';
	arSystemStateNames[104] :='Group4_L2_f';
	arSystemStateNames[105] :='Group4_L3_f';
	arSystemStateNames[106] :='Group4_3F_E';
	arSystemStateNames[107] :='Group4_3F_Field_Rotation';
	arSystemStateNames[108] :='Group4_3F_E_Reactive';
	arSystemStateNames[109] :='Group5_L1_P';
	arSystemStateNames[110] :='Group5_L2_P';
	arSystemStateNames[111] :='Group5_L3_P';
	arSystemStateNames[112] :='Group5_L1_Q';
	arSystemStateNames[113] :='Group5_L2_Q';
	arSystemStateNames[114] :='Group5_L3_Q';
	arSystemStateNames[115] :='Group5_L1_V';
	arSystemStateNames[116] :='Group5_L2_V';
	arSystemStateNames[117] :='Group5_L3_V';
	arSystemStateNames[118] :='Group5_L1_I';
	arSystemStateNames[119] :='Group5_L2_I';
	arSystemStateNames[120] :='Group5_L3_I';
	arSystemStateNames[121] :='Group5_L1_f';
	arSystemStateNames[122] :='Group5_L2_f';
	arSystemStateNames[123] :='Group5_L3_f';
	arSystemStateNames[124] :='Group5_3F_E';
	arSystemStateNames[125] :='Group5_3F_Field_Rotation';
	arSystemStateNames[126] :='Group5_3F_E_Reactive';
	arSystemStateNames[127] :='Group6_L1_P';
	arSystemStateNames[128] :='Group6_L2_P';
	arSystemStateNames[129] :='Group6_L3_P';
	arSystemStateNames[130] :='Group6_L1_Q';
	arSystemStateNames[131] :='Group6_L2_Q';
	arSystemStateNames[132] :='Group6_L3_Q';
	arSystemStateNames[133] :='Group6_L1_V';
	arSystemStateNames[134] :='Group6_L2_V';
	arSystemStateNames[135] :='Group6_L3_V';
	arSystemStateNames[136] :='Group6_L1_I';
	arSystemStateNames[137] :='Group6_L2_I';
	arSystemStateNames[138] :='Group6_L3_I';
	arSystemStateNames[139] :='Group6_L1_f';
	arSystemStateNames[140] :='Group6_L2_f';
	arSystemStateNames[141] :='Group6_L3_f';
	arSystemStateNames[142] :='Group6_3F_E';
	arSystemStateNames[143] :='Group6_3F_Field_Rotation';
	arSystemStateNames[144] :='Group6_3F_E_Reactive';
	arSystemStateNames[145] :='Group7_L1_P';
	arSystemStateNames[146] :='Group7_L2_P';
	arSystemStateNames[147] :='Group7_L3_P';
	arSystemStateNames[148] :='Group7_L1_Q';
	arSystemStateNames[149] :='Group7_L2_Q';
	arSystemStateNames[150] :='Group7_L3_Q';
	arSystemStateNames[151] :='Group7_L1_V';
	arSystemStateNames[152] :='Group7_L2_V';
	arSystemStateNames[153] :='Group7_L3_V';
	arSystemStateNames[154] :='Group7_L1_I';
	arSystemStateNames[155] :='Group7_L2_I';
	arSystemStateNames[156] :='Group7_L3_I';
	arSystemStateNames[157] :='Group7_L1_f';
	arSystemStateNames[158] :='Group7_L2_f';
	arSystemStateNames[159] :='Group7_L3_f';
	arSystemStateNames[160] :='Group7_3F_E';
	arSystemStateNames[161] :='Group7_3F_Field_Rotation';
	arSystemStateNames[162] :='Group7_3F_E_Reactive';
	arSystemStateNames[163] :='Group8_L1_P';
	arSystemStateNames[164] :='Group8_L2_P';
	arSystemStateNames[165] :='Group8_L3_P';
	arSystemStateNames[166] :='Group8_L1_Q';
	arSystemStateNames[167] :='Group8_L2_Q';
	arSystemStateNames[168] :='Group8_L3_Q';
	arSystemStateNames[169] :='Group8_L1_V';
	arSystemStateNames[170] :='Group8_L2_V';
	arSystemStateNames[171] :='Group8_L3_V';
	arSystemStateNames[172] :='Group8_L1_I';
	arSystemStateNames[173] :='Group8_L2_I';
	arSystemStateNames[174] :='Group8_L3_I';
	arSystemStateNames[175] :='Group8_L1_f';
	arSystemStateNames[176] :='Group8_L2_f';
	arSystemStateNames[177] :='Group8_L3_f';
	arSystemStateNames[178] :='Group8_3F_E';
	arSystemStateNames[179] :='Group8_3F_Field_Rotation';
	arSystemStateNames[180] :='Group8_3F_E_Reactive';
	arSystemStateNames[181] :='Group9_L1_P';
	arSystemStateNames[182] :='Group9_L2_P';
	arSystemStateNames[183] :='Group9_L3_P';
	arSystemStateNames[184] :='Group9_L1_Q';
	arSystemStateNames[185] :='Group9_L2_Q';
	arSystemStateNames[186] :='Group9_L3_Q';
	arSystemStateNames[187] :='Group9_L1_V';
	arSystemStateNames[188] :='Group9_L2_V';
	arSystemStateNames[189] :='Group9_L3_V';
	arSystemStateNames[190] :='Group9_L1_I';
	arSystemStateNames[191] :='Group9_L2_I';
	arSystemStateNames[192] :='Group9_L3_I';
	arSystemStateNames[193] :='Group9_L1_f';
	arSystemStateNames[194] :='Group9_L2_f';
	arSystemStateNames[195] :='Group9_L3_f';
	arSystemStateNames[196] :='Group9_3F_E';
	arSystemStateNames[197] :='Group9_3F_Field_Rotation';
	arSystemStateNames[198] :='Group9_3F_E_Reactive';
	arSystemStateNames[199] :='Bus_Connector_L1_P';
	arSystemStateNames[200] :='Bus_Connector_L2_P';
	arSystemStateNames[201] :='Bus_Connector_L3_P';
	arSystemStateNames[202] :='Bus_Connector_L1_Q';
	arSystemStateNames[203] :='Bus_Connector_L2_Q';
	arSystemStateNames[204] :='Bus_Connector_L3_Q';
	arSystemStateNames[205] :='Bus_Connector_L1_V';
	arSystemStateNames[206] :='Bus_Connector_L2_V';
	arSystemStateNames[207] :='Bus_Connector_L3_V';
	arSystemStateNames[208] :='Bus_Connector_L1_I';
	arSystemStateNames[209] :='Bus_Connector_L2_I';
	arSystemStateNames[210] :='Bus_Connector_L3_I';
	arSystemStateNames[211] :='Bus_Connector_L1_f';
	arSystemStateNames[212] :='Bus_Connector_L2_f';
	arSystemStateNames[213] :='Bus_Connector_L3_f';
	arSystemStateNames[214] :='Bus_Connector_3F_radians';
	arSystemStateNames[215] :='Bus_Connector_3F_Sync_close_requested';
	arSystemStateNames[216] :='Bus_Connector_3F_Sync_closed';
	arSystemStateNames[217] :='Bus_Connector_3F_Sync_close_requested_panel';
	arSystemStateNames[218] :='Bus_Connector_3F_Sync_denied_panel';
	arSystemStateNames[219] :='Bus_Connector_3F_Sync_close_requested_modbus';
	arSystemStateNames[220] :='Bus_Connector_3F_Sync_denied_modbus';
	arSystemStateNames[221] :='Bus_Connector_3F_Field_Rotation';
	arSystemStateNames[222] :='CHP_control_grid_bus_select_controlswitch';
	arSystemStateNames[223] :='CHP_control_baterry_bus_select_controlswitch';
	arSystemStateNames[224] :='CHP_control_auto_bus_select_controlswitch';
	arSystemStateNames[225] :='CHP_control_Offgrid_request';
	arSystemStateNames[226] :='CHP_control_Offgrid_Active_Power_control';
	arSystemStateNames[227] :='CHP_control_internal_contacter_switch_state';
	arSystemStateNames[228] :='EV_control_control_signal';
	arSystemStateNames[229] :='Mixer_control_control_signal';
	arSystemStateNames[230] :='Group1_3F_Auto_relay_control_battery_bus';
	arSystemStateNames[231] :='Group1_3F_Auto_relay_control_grid_bus';
	arSystemStateNames[232] :='Group1_3F_Selector_auto_bus_select';
	arSystemStateNames[233] :='Group1_3F_relay_state_battery_bus';
	arSystemStateNames[234] :='Group1_3F_relay_state_grid_bus';
	arSystemStateNames[233] :='Group2_3F_Auto_relay_control_battery_bus';
	arSystemStateNames[234] :='Group2_3F_Auto_relay_control_grid_bus';
	arSystemStateNames[235] :='Group2_3F_Selector_auto_bus_select';
	arSystemStateNames[236] :='Group2_3F_relay_state_battery_bus';
	arSystemStateNames[237] :='Group2_3F_relay_state_grid_bus';
	arSystemStateNames[236] :='Group3_3F_Auto_relay_control_battery_bus';
	arSystemStateNames[237] :='Group3_3F_Auto_relay_control_grid_bus';
	arSystemStateNames[238] :='Group3_3F_Selector_auto_bus_select';
	arSystemStateNames[239] :='Group3_3F_relay_state_battery_bus';
	arSystemStateNames[240] :='Group3_3F_relay_state_grid_bus';
	arSystemStateNames[239] :='Group4_3F_Auto_relay_control_battery_bus';
	arSystemStateNames[240] :='Group4_3F_Auto_relay_control_grid_bus';
	arSystemStateNames[241] :='Group4_3F_Selector_auto_bus_select';
	arSystemStateNames[242] :='Group4_3F_relay_state_battery_bus';
	arSystemStateNames[243] :='Group4_3F_relay_state_grid_bus';
	arSystemStateNames[242] :='Group5_3F_Auto_relay_control_battery_bus';
	arSystemStateNames[243] :='Group5_3F_Auto_relay_control_grid_bus';
	arSystemStateNames[244] :='Group5_3F_Selector_auto_bus_select';
	arSystemStateNames[245] :='Group5_3F_relay_state_battery_bus';
	arSystemStateNames[246] :='Group5_3F_relay_state_grid_bus';
	arSystemStateNames[245] :='Group6_3F_Auto_relay_control_battery_bus';
	arSystemStateNames[246] :='Group6_3F_Auto_relay_control_grid_bus';
	arSystemStateNames[247] :='Group6_3F_Selector_auto_bus_select';
	arSystemStateNames[248] :='Group6_3F_relay_state_battery_bus';
	arSystemStateNames[249] :='Group6_3F_relay_state_grid_bus';
	arSystemStateNames[248] :='Group7_3F_Auto_relay_control_battery_bus';
	arSystemStateNames[249] :='Group7_3F_Auto_relay_control_grid_bus';
	arSystemStateNames[250] :='Group7_3F_Selector_auto_bus_select';
	arSystemStateNames[251] :='Group7_3F_relay_state_battery_bus';
	arSystemStateNames[252] :='Group7_3F_relay_state_grid_bus';
	arSystemStateNames[251] :='Group8_3F_Auto_relay_control_battery_bus';
	arSystemStateNames[252] :='Group8_3F_Auto_relay_control_grid_bus';
	arSystemStateNames[253] :='Group8_3F_Selector_auto_bus_select';
	arSystemStateNames[254] :='Group8_3F_relay_state_battery_bus';
	arSystemStateNames[255] :='Group8_3F_relay_state_grid_bus';
	arSystemStateNames[256] :='Group9_3F_Auto_relay_control_battery_bus';
	arSystemStateNames[257] :='Group9_3F_Auto_relay_control_grid_bus';
	arSystemStateNames[258] :='Group9_3F_Selector_auto_bus_select';
	arSystemStateNames[259] :='Group9_3F_relay_state_battery_bus';
	arSystemStateNames[260] :='Group9_3F_relay_state_grid_bus';
	arSystemStateNames[261] :='Group_control_Frequencybased_bus_selecting_state';
	arSystemStateNames[262] :='Group_control_min_time_above_switch_frequency';
	arSystemStateNames[263] :='Group_control_min_time_below_switch_frequency';
	arSystemStateNames[264] :='Group1_3F_Switch_frequency_to_batterybus';
	arSystemStateNames[265] :='Group1_3F_Switch_frequency_to_gridbus';
	arSystemStateNames[266] :='Group1_3F_min_time_between_switching';
	arSystemStateNames[267] :='Group2_3F_Switch_frequency_to_batterybus';
	arSystemStateNames[268] :='Group2_3F_Switch_frequency_to_gridbus';
	arSystemStateNames[269] :='Group2_3F_min_time_between_switching';
	arSystemStateNames[268] :='Group3_3F_Switch_frequency_to_batterybus';
	arSystemStateNames[269] :='Group3_3F_Switch_frequency_to_gridbus';
	arSystemStateNames[270] :='Group3_3F_min_time_between_switching';
	arSystemStateNames[271] :='Group4_3F_Switch_frequency_to_batterybus';
	arSystemStateNames[270] :='Group4_3F_Switch_frequency_to_gridbus';
	arSystemStateNames[271] :='Group4_3F_min_time_between_switching';
	arSystemStateNames[272] :='Group5_3F_Switch_frequency_to_batterybus';
	arSystemStateNames[273] :='Group5_3F_Switch_frequency_to_gridbus';
	arSystemStateNames[272] :='Group5_3F_min_time_between_switching';
	arSystemStateNames[273] :='Group6_3F_Switch_frequency_to_batterybus';
	arSystemStateNames[274] :='Group6_3F_Switch_frequency_to_gridbus';
	arSystemStateNames[275] :='Group6_3F_min_time_between_switching';
	arSystemStateNames[274] :='Group7_3F_Switch_frequency_to_batterybus';
	arSystemStateNames[275] :='Group7_3F_Switch_frequency_to_gridbus';
	arSystemStateNames[276] :='Group7_3F_min_time_between_switching';
	arSystemStateNames[277] :='Group8_3F_Switch_frequency_to_batterybus';
	arSystemStateNames[276] :='Group8_3F_Switch_frequency_to_gridbus';
	arSystemStateNames[277] :='Group8_3F_min_time_between_switching';
	arSystemStateNames[278] :='Group9_3F_Switch_frequency_to_batterybus';
	arSystemStateNames[279] :='Group9_3F_Switch_frequency_to_gridbus';
	arSystemStateNames[278] :='Group9_3F_min_time_between_switching';
	arSystemStateNames[279] :='Control_panel_status_warning_led';
	arSystemStateNames[280] :='Control_panel_status_error_led';
	arSystemStateNames[281] :='Control_panel_status_operational_led';
END_PROGRAM

(* POU 04. Frequency based Bus Select/run_group_switching, ST *)
PROGRAM run_group_switching
VAR
(*
	Group1 :fbSwitchRelaysBatOrGridBus; (* CHP Group has special rules *)
	Group2 :fbSwitchRelaysBatOrGridBus; (*  *)
	Group3 :fbSwitchRelaysBatOrGridBus; (*  *)
	Group4 :fbSwitchRelaysBatOrGridBus; (*  *)
	Group5 :fbSwitchRelaysBatOrGridBus; (*  *)
	Group6 :fbSwitchRelaysBatOrGridBus; (*  *)
	Group7 :fbSwitchRelaysBatOrGridBus; (*  *)
	Group8 :fbSwitchRelaysBatOrGridBus; (*  *)
	Group9 :fbSwitchRelaysBatOrGridBus; (*  *)
*)
	y: INT;
END_VAR
(* frequency based switching is deactivated BY default AND can be activated via modbus *)

	Group_control_Frequencybased_bus_selecting_state := REAL_TO_BOOL(arSystemState[275]) ;

	(* default switching gap time is 2000ms and can never be set lower than 1000ms via Modbus *)
	(*Switch_Gap_Time								:= REAL_TO_INT(arSystemState[99]);*)
	IF Switch_Gap_Time < 10 THEN
		Switch_Gap_Time := 10;
	END_IF

IF Group_control_Frequencybased_bus_selecting_state = TRUE THEN
	Group1();
	CHP_switch_delay();
	Group2();
	Group3();
	Group4();
	Group5();
	Group6();
	Group7();
	Group8();
	Group9();
END_IF
END_PROGRAM

(* POU 04. Frequency based Bus Select/CHP_switch_delay, ST *)
PROGRAM CHP_switch_delay
(* ____________________________  USED GLOBAL VARIABLES  ___________________________

VAR_INPUT

	CHP_new_state_grid_bus							:	BOOL; (* request based on frequency *)
	CHP_new_state_battery_bus						:	BOOL; (* request based on frequency *)

	CHP_relay_state_battery_bus   							AT %IX134.1  : BOOL;  (* INVERTED INPUTS *)
	CHP_relay_state_grid_bus   								AT %IX134.2  : BOOL;  (* INVERTED INPUTS *)
	
	CHP_control_internal_contacter_switch_state

END_VAR

VAR_OUTPUT

	Group1_3F_Auto_relay_control_battery_bus							:	BOOL; (* request based on frequency, has delayed switching!! *)
	Group1_3F_Auto_relay_control_battery_bus							:	BOOL; (* request based on frequency, has delayed switching!! *)

END_VAR
*)

VAR
	y: BOOL :=FALSE;
	z: INT;
END_VAR
(* CHP handler uses frequency based switching input to control real CHP swithcing when auto input is high *)
(* CHP handler delays switching, such that the CHP can depower and disconnect before switch *)
(* CHP handler delays on-switching, making sure the CHP is disconnected. *)
(* CHP handler delays on-switching, making sure the CHP will connect to the right bus (in the right mode). *)

(* ____________________________  AUTO SWITCH CONTROL  ___________________________ *)
IF Group1_3F_Selector_auto_bus_select = TRUE THEN
	z := z + 1;
	(*check if wanted state to CHP signal is right, change when required *)
	IF CHP_new_state_grid_bus =TRUE THEN
		CHP_control_Offgrid_request :=FALSE;
		z :=0;
		y := FALSE;
	ELSE
		IF CHP_new_state_battery_bus = TRUE THEN
		CHP_control_Offgrid_request :=TRUE;
		z := 100;
		y := TRUE;
		END_IF;
	END_IF;

	(* perform switch between busses when CHP has disconnceted *)
	IF CHP_control_internal_contacter_switch_state = FALSE THEN

		(* Close bat relais when grid relais is open en bat request is still true*)
		IF CHP_new_state_battery_bus =TRUE  THEN

			IF CHP_relay_state_grid_bus = TRUE THEN (* INVERTED INPUTS *)
				Group1_3F_Auto_relay_control_battery_bus := TRUE;
			END_IF;
			Group1_3F_Auto_relay_control_grid_bus := FALSE; (* Disconnect GRID SCWICH*)
		END_IF;

		(* Close grid relais when bat relais is open en grid request is still true*)
		IF CHP_new_state_grid_bus =TRUE  THEN

			IF CHP_relay_state_battery_bus = TRUE THEN (* INVERTED INPUTS *)
				Group1_3F_Auto_relay_control_grid_bus := TRUE;
			END_IF;
			Group1_3F_Auto_relay_control_battery_bus := FALSE; (* Disconnect *)
		END_IF;
	END_IF;


(* ____________________________  MANUAL CONTROL  ___________________________ *)
ELSE
	z := 200;
	(* check if batbus relais is closed, if so, request offgrid (via wanted state *)
	IF Group1_3F_relay_state_battery_bus = TRUE THEN
		CHP_control_Offgrid_request :=TRUE;
	ELSE (* IF Group1_3F_relay_state_grid_bus THEN *)
		CHP_control_Offgrid_request :=FALSE;
	END_IF;

	Group1_3F_Auto_relay_control_grid_bus := FALSE; (* Disconnect GRID SCWICH*)
	Group1_3F_Auto_relay_control_battery_bus := FALSE; (* Disconnect *)
END_IF;
END_PROGRAM

(* POU 04. Frequency based Bus Select/Group2, FBD *)
PROGRAM Group2
VAR
	Switch:Auto_switch_new;
	request_grid: BOOL;
	request_testbus: BOOL;
	Delayer: Auto_delayer;
END_VAR
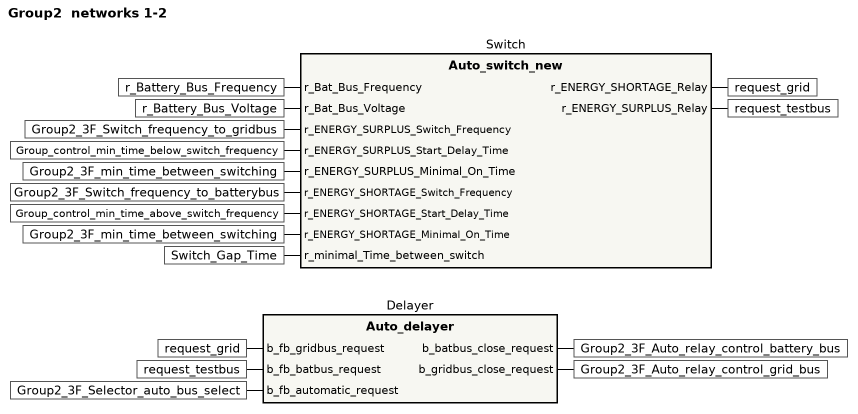
_FBD_ (* Function Block Diagram *)
NETWORK 1
	Switch:Auto_switch_new(r_Bat_Bus_Frequency: r_Battery_Bus_Frequency, r_Bat_Bus_Voltage: r_Battery_Bus_Voltage, r_ENERGY_SURPLUS_Switch_Frequency: Group2_3F_Switch_frequency_to_gridbus, r_ENERGY_SURPLUS_Start_Delay_Time: Group_control_min_time_below_switch_frequency, r_ENERGY_SURPLUS_Minimal_On_Time: Group2_3F_min_time_between_switching, r_ENERGY_SHORTAGE_Switch_Frequency: Group2_3F_Switch_frequency_to_batterybus, r_ENERGY_SHORTAGE_Start_Delay_Time: Group_control_min_time_above_switch_frequency, r_ENERGY_SHORTAGE_Minimal_On_Time: Group2_3F_min_time_between_switching, r_minimal_Time_between_switch: Switch_Gap_Time, r_ENERGY_SURPLUS_Relay => request_testbus) => request_grid
NETWORK 2
	Delayer:Auto_delayer(b_fb_gridbus_request: request_grid, b_fb_batbus_request: request_testbus, b_fb_automatic_request: Group2_3F_Selector_auto_bus_select, b_gridbus_close_request => Group2_3F_Auto_relay_control_grid_bus) => Group2_3F_Auto_relay_control_battery_bus
_END_FBD_
(* the same logic as Structured Text *)
(* Network 1 *)
Switch(r_Bat_Bus_Frequency := r_Battery_Bus_Frequency, r_Bat_Bus_Voltage := r_Battery_Bus_Voltage, r_ENERGY_SURPLUS_Switch_Frequency := Group2_3F_Switch_frequency_to_gridbus, r_ENERGY_SURPLUS_Start_Delay_Time := Group_control_min_time_below_switch_frequency, r_ENERGY_SURPLUS_Minimal_On_Time := Group2_3F_min_time_between_switching, r_ENERGY_SHORTAGE_Switch_Frequency := Group2_3F_Switch_frequency_to_batterybus, r_ENERGY_SHORTAGE_Start_Delay_Time := Group_control_min_time_above_switch_frequency, r_ENERGY_SHORTAGE_Minimal_On_Time := Group2_3F_min_time_between_switching, r_minimal_Time_between_switch := Switch_Gap_Time);
request_testbus := Switch.r_ENERGY_SURPLUS_Relay;
request_grid := Switch.r_ENERGY_SHORTAGE_Relay;
(* Network 2 *)
Delayer(b_fb_gridbus_request := request_grid, b_fb_batbus_request := request_testbus, b_fb_automatic_request := Group2_3F_Selector_auto_bus_select);
Group2_3F_Auto_relay_control_grid_bus := Delayer.b_gridbus_close_request;
Group2_3F_Auto_relay_control_battery_bus := Delayer.b_batbus_close_request;
END_PROGRAM

(* POU 04. Frequency based Bus Select/Auto_delayer, ST *)
FUNCTION_BLOCK Auto_delayer

VAR_INPUT

	b_fb_gridbus_request							:	BOOL; (* request based on frequency, has no delayed switching!! *)
	b_fb_batbus_request								:	BOOL; (* request based on frequency, has no delayed switching!! *)
	b_fb_automatic_request							:	BOOL; (* request based on frequency, has delayed switching!! *)

END_VAR

VAR_OUTPUT

	b_batbus_close_request							:	BOOL; (* request based on frequency, has delayed switching!! *)
	b_gridbus_close_request						:	BOOL; (* request based on frequency, has delayed switching!! *)

END_VAR
VAR

END_VAR
IF b_fb_automatic_request = TRUE THEN

	(* perform switch between busses when both hav disconnceted *)
	IF b_fb_gridbus_request = TRUE THEN
		(* Close grid relais when bat relais is open en grid request is still true*)
		IF b_batbus_close_request = TRUE  THEN
			b_batbus_close_request := FALSE; (* Disconnect BAT SCWICH*)
		ELSE
			b_gridbus_close_request := TRUE;
		END_IF;

		(* Close bat relais when grid relais is open en bat request is still true*)
	ELSIF b_fb_batbus_request = TRUE THEN
		IF b_gridbus_close_request = TRUE THEN
			b_gridbus_close_request := FALSE;
		ELSE
			b_batbus_close_request := TRUE;
		END_IF;
	END_IF;
(* ____________________________  MANUAL CONTROL  ___________________________ *)
ELSE
	(* check if batbus relais is closed, if so, request offgrid (via wanted state *)
		b_batbus_close_request :=FALSE;
		b_gridbus_close_request :=FALSE;
END_IF;
END_FUNCTION_BLOCK

(* POU 04. Frequency based Bus Select/Group3, FBD *)
PROGRAM Group3
VAR

	request_grid: BOOL;
	request_testbus: BOOL;
	Delayer: Auto_delayer;
	Switch: Auto_switch_new;
END_VAR
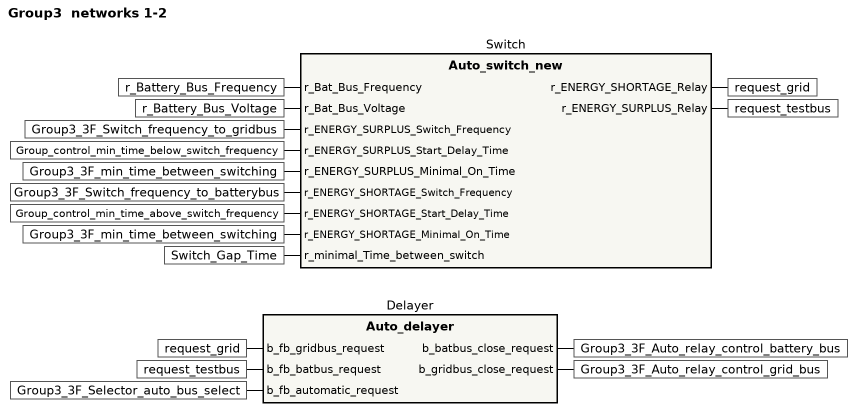
_FBD_ (* Function Block Diagram *)
NETWORK 1
	Switch:Auto_switch_new(r_Bat_Bus_Frequency: r_Battery_Bus_Frequency, r_Bat_Bus_Voltage: r_Battery_Bus_Voltage, r_ENERGY_SURPLUS_Switch_Frequency: Group3_3F_Switch_frequency_to_gridbus, r_ENERGY_SURPLUS_Start_Delay_Time: Group_control_min_time_below_switch_frequency, r_ENERGY_SURPLUS_Minimal_On_Time: Group3_3F_min_time_between_switching, r_ENERGY_SHORTAGE_Switch_Frequency: Group3_3F_Switch_frequency_to_batterybus, r_ENERGY_SHORTAGE_Start_Delay_Time: Group_control_min_time_above_switch_frequency, r_ENERGY_SHORTAGE_Minimal_On_Time: Group3_3F_min_time_between_switching, r_minimal_Time_between_switch: Switch_Gap_Time, r_ENERGY_SURPLUS_Relay => request_testbus) => request_grid
NETWORK 2
	Delayer:Auto_delayer(b_fb_gridbus_request: request_grid, b_fb_batbus_request: request_testbus, b_fb_automatic_request: Group3_3F_Selector_auto_bus_select, b_gridbus_close_request => Group3_3F_Auto_relay_control_grid_bus) => Group3_3F_Auto_relay_control_battery_bus
_END_FBD_
(* the same logic as Structured Text *)
(* Network 1 *)
Switch(r_Bat_Bus_Frequency := r_Battery_Bus_Frequency, r_Bat_Bus_Voltage := r_Battery_Bus_Voltage, r_ENERGY_SURPLUS_Switch_Frequency := Group3_3F_Switch_frequency_to_gridbus, r_ENERGY_SURPLUS_Start_Delay_Time := Group_control_min_time_below_switch_frequency, r_ENERGY_SURPLUS_Minimal_On_Time := Group3_3F_min_time_between_switching, r_ENERGY_SHORTAGE_Switch_Frequency := Group3_3F_Switch_frequency_to_batterybus, r_ENERGY_SHORTAGE_Start_Delay_Time := Group_control_min_time_above_switch_frequency, r_ENERGY_SHORTAGE_Minimal_On_Time := Group3_3F_min_time_between_switching, r_minimal_Time_between_switch := Switch_Gap_Time);
request_testbus := Switch.r_ENERGY_SURPLUS_Relay;
request_grid := Switch.r_ENERGY_SHORTAGE_Relay;
(* Network 2 *)
Delayer(b_fb_gridbus_request := request_grid, b_fb_batbus_request := request_testbus, b_fb_automatic_request := Group3_3F_Selector_auto_bus_select);
Group3_3F_Auto_relay_control_grid_bus := Delayer.b_gridbus_close_request;
Group3_3F_Auto_relay_control_battery_bus := Delayer.b_batbus_close_request;
END_PROGRAM

(* POU 04. Frequency based Bus Select/Group4, FBD *)
PROGRAM Group4
VAR

	request_grid: BOOL;
	request_testbus: BOOL;
	Delayer: Auto_delayer;
	Switch: Auto_switch_new;
END_VAR
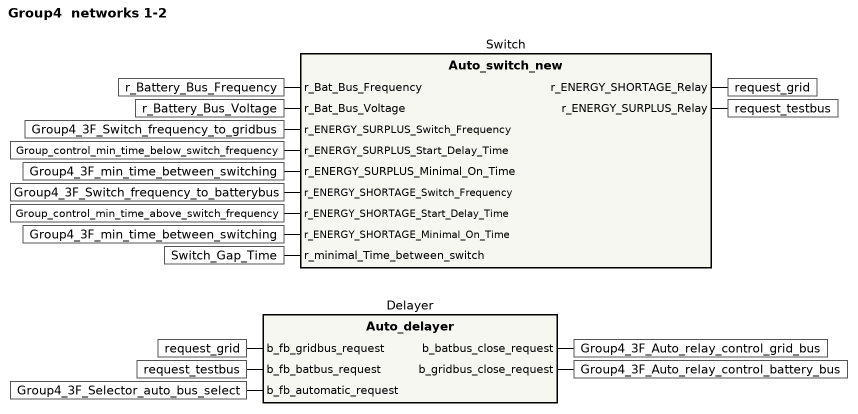
_FBD_ (* Function Block Diagram *)
NETWORK 1
	Switch:Auto_switch_new(r_Bat_Bus_Frequency: r_Battery_Bus_Frequency, r_Bat_Bus_Voltage: r_Battery_Bus_Voltage, r_ENERGY_SURPLUS_Switch_Frequency: Group4_3F_Switch_frequency_to_gridbus, r_ENERGY_SURPLUS_Start_Delay_Time: Group_control_min_time_below_switch_frequency, r_ENERGY_SURPLUS_Minimal_On_Time: Group4_3F_min_time_between_switching, r_ENERGY_SHORTAGE_Switch_Frequency: Group4_3F_Switch_frequency_to_batterybus, r_ENERGY_SHORTAGE_Start_Delay_Time: Group_control_min_time_above_switch_frequency, r_ENERGY_SHORTAGE_Minimal_On_Time: Group4_3F_min_time_between_switching, r_minimal_Time_between_switch: Switch_Gap_Time, r_ENERGY_SURPLUS_Relay => request_testbus) => request_grid
NETWORK 2
	Delayer:Auto_delayer(b_fb_gridbus_request: request_grid, b_fb_batbus_request: request_testbus, b_fb_automatic_request: Group4_3F_Selector_auto_bus_select, b_gridbus_close_request => Group4_3F_Auto_relay_control_battery_bus) => Group4_3F_Auto_relay_control_grid_bus
_END_FBD_
(* the same logic as Structured Text *)
(* Network 1 *)
Switch(r_Bat_Bus_Frequency := r_Battery_Bus_Frequency, r_Bat_Bus_Voltage := r_Battery_Bus_Voltage, r_ENERGY_SURPLUS_Switch_Frequency := Group4_3F_Switch_frequency_to_gridbus, r_ENERGY_SURPLUS_Start_Delay_Time := Group_control_min_time_below_switch_frequency, r_ENERGY_SURPLUS_Minimal_On_Time := Group4_3F_min_time_between_switching, r_ENERGY_SHORTAGE_Switch_Frequency := Group4_3F_Switch_frequency_to_batterybus, r_ENERGY_SHORTAGE_Start_Delay_Time := Group_control_min_time_above_switch_frequency, r_ENERGY_SHORTAGE_Minimal_On_Time := Group4_3F_min_time_between_switching, r_minimal_Time_between_switch := Switch_Gap_Time);
request_testbus := Switch.r_ENERGY_SURPLUS_Relay;
request_grid := Switch.r_ENERGY_SHORTAGE_Relay;
(* Network 2 *)
Delayer(b_fb_gridbus_request := request_grid, b_fb_batbus_request := request_testbus, b_fb_automatic_request := Group4_3F_Selector_auto_bus_select);
Group4_3F_Auto_relay_control_battery_bus := Delayer.b_gridbus_close_request;
Group4_3F_Auto_relay_control_grid_bus := Delayer.b_batbus_close_request;
END_PROGRAM

(* POU 04. Frequency based Bus Select/Group5, FBD *)
PROGRAM Group5
VAR

	request_grid: BOOL;
	request_testbus: BOOL;
	Delayer: Auto_delayer;
	Switch: Auto_switch_new;
END_VAR
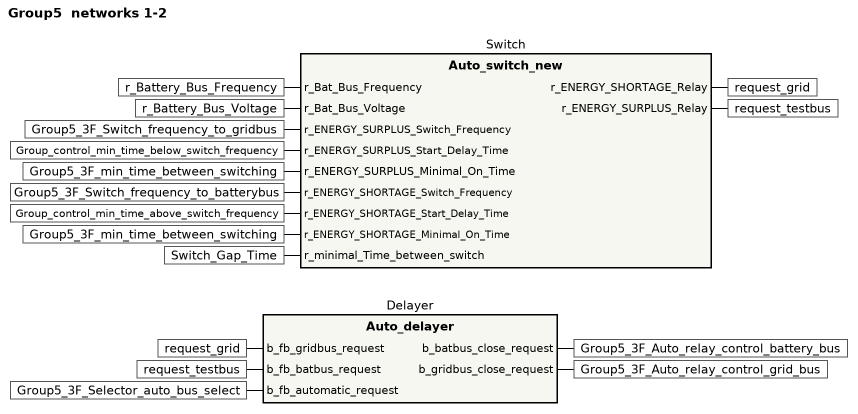
_FBD_ (* Function Block Diagram *)
NETWORK 1
	Switch:Auto_switch_new(r_Bat_Bus_Frequency: r_Battery_Bus_Frequency, r_Bat_Bus_Voltage: r_Battery_Bus_Voltage, r_ENERGY_SURPLUS_Switch_Frequency: Group5_3F_Switch_frequency_to_gridbus, r_ENERGY_SURPLUS_Start_Delay_Time: Group_control_min_time_below_switch_frequency, r_ENERGY_SURPLUS_Minimal_On_Time: Group5_3F_min_time_between_switching, r_ENERGY_SHORTAGE_Switch_Frequency: Group5_3F_Switch_frequency_to_batterybus, r_ENERGY_SHORTAGE_Start_Delay_Time: Group_control_min_time_above_switch_frequency, r_ENERGY_SHORTAGE_Minimal_On_Time: Group5_3F_min_time_between_switching, r_minimal_Time_between_switch: Switch_Gap_Time, r_ENERGY_SURPLUS_Relay => request_testbus) => request_grid
NETWORK 2
	Delayer:Auto_delayer(b_fb_gridbus_request: request_grid, b_fb_batbus_request: request_testbus, b_fb_automatic_request: Group5_3F_Selector_auto_bus_select, b_gridbus_close_request => Group5_3F_Auto_relay_control_grid_bus) => Group5_3F_Auto_relay_control_battery_bus
_END_FBD_
(* the same logic as Structured Text *)
(* Network 1 *)
Switch(r_Bat_Bus_Frequency := r_Battery_Bus_Frequency, r_Bat_Bus_Voltage := r_Battery_Bus_Voltage, r_ENERGY_SURPLUS_Switch_Frequency := Group5_3F_Switch_frequency_to_gridbus, r_ENERGY_SURPLUS_Start_Delay_Time := Group_control_min_time_below_switch_frequency, r_ENERGY_SURPLUS_Minimal_On_Time := Group5_3F_min_time_between_switching, r_ENERGY_SHORTAGE_Switch_Frequency := Group5_3F_Switch_frequency_to_batterybus, r_ENERGY_SHORTAGE_Start_Delay_Time := Group_control_min_time_above_switch_frequency, r_ENERGY_SHORTAGE_Minimal_On_Time := Group5_3F_min_time_between_switching, r_minimal_Time_between_switch := Switch_Gap_Time);
request_testbus := Switch.r_ENERGY_SURPLUS_Relay;
request_grid := Switch.r_ENERGY_SHORTAGE_Relay;
(* Network 2 *)
Delayer(b_fb_gridbus_request := request_grid, b_fb_batbus_request := request_testbus, b_fb_automatic_request := Group5_3F_Selector_auto_bus_select);
Group5_3F_Auto_relay_control_grid_bus := Delayer.b_gridbus_close_request;
Group5_3F_Auto_relay_control_battery_bus := Delayer.b_batbus_close_request;
END_PROGRAM

(* POU 04. Frequency based Bus Select/Group6, FBD *)
PROGRAM Group6
VAR
	Switch:Auto_switch_new;
	request_grid:BOOL := TRUE;
	request_testbus:BOOL := FALSE;
	Delayer: Auto_delayer;
END_VAR
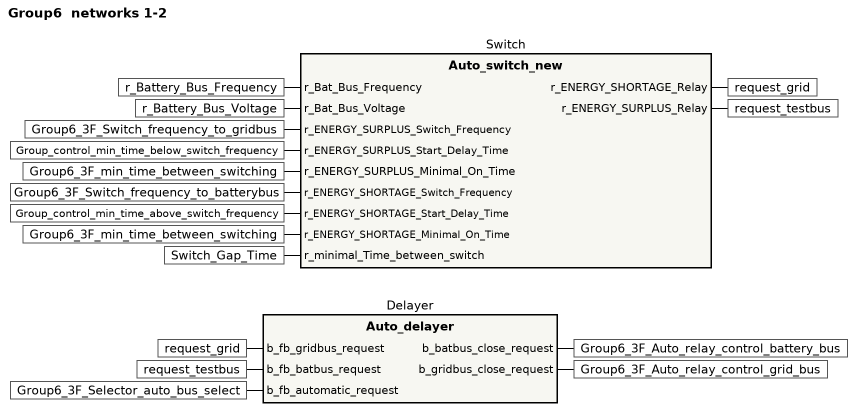
_FBD_ (* Function Block Diagram *)
NETWORK 1
	Switch:Auto_switch_new(r_Bat_Bus_Frequency: r_Battery_Bus_Frequency, r_Bat_Bus_Voltage: r_Battery_Bus_Voltage, r_ENERGY_SURPLUS_Switch_Frequency: Group6_3F_Switch_frequency_to_gridbus, r_ENERGY_SURPLUS_Start_Delay_Time: Group_control_min_time_below_switch_frequency, r_ENERGY_SURPLUS_Minimal_On_Time: Group6_3F_min_time_between_switching, r_ENERGY_SHORTAGE_Switch_Frequency: Group6_3F_Switch_frequency_to_batterybus, r_ENERGY_SHORTAGE_Start_Delay_Time: Group_control_min_time_above_switch_frequency, r_ENERGY_SHORTAGE_Minimal_On_Time: Group6_3F_min_time_between_switching, r_minimal_Time_between_switch: Switch_Gap_Time, r_ENERGY_SURPLUS_Relay => request_testbus) => request_grid
NETWORK 2
	Delayer:Auto_delayer(b_fb_gridbus_request: request_grid, b_fb_batbus_request: request_testbus, b_fb_automatic_request: Group6_3F_Selector_auto_bus_select, b_gridbus_close_request => Group6_3F_Auto_relay_control_grid_bus) => Group6_3F_Auto_relay_control_battery_bus
_END_FBD_
(* the same logic as Structured Text *)
(* Network 1 *)
Switch(r_Bat_Bus_Frequency := r_Battery_Bus_Frequency, r_Bat_Bus_Voltage := r_Battery_Bus_Voltage, r_ENERGY_SURPLUS_Switch_Frequency := Group6_3F_Switch_frequency_to_gridbus, r_ENERGY_SURPLUS_Start_Delay_Time := Group_control_min_time_below_switch_frequency, r_ENERGY_SURPLUS_Minimal_On_Time := Group6_3F_min_time_between_switching, r_ENERGY_SHORTAGE_Switch_Frequency := Group6_3F_Switch_frequency_to_batterybus, r_ENERGY_SHORTAGE_Start_Delay_Time := Group_control_min_time_above_switch_frequency, r_ENERGY_SHORTAGE_Minimal_On_Time := Group6_3F_min_time_between_switching, r_minimal_Time_between_switch := Switch_Gap_Time);
request_testbus := Switch.r_ENERGY_SURPLUS_Relay;
request_grid := Switch.r_ENERGY_SHORTAGE_Relay;
(* Network 2 *)
Delayer(b_fb_gridbus_request := request_grid, b_fb_batbus_request := request_testbus, b_fb_automatic_request := Group6_3F_Selector_auto_bus_select);
Group6_3F_Auto_relay_control_grid_bus := Delayer.b_gridbus_close_request;
Group6_3F_Auto_relay_control_battery_bus := Delayer.b_batbus_close_request;
END_PROGRAM

(* POU 04. Frequency based Bus Select/Group7, FBD *)
PROGRAM Group7
VAR

	request_grid: BOOL;
	request_testbus: BOOL;
	Delayer: Auto_delayer;
	Switch: Auto_switch_new;
END_VAR
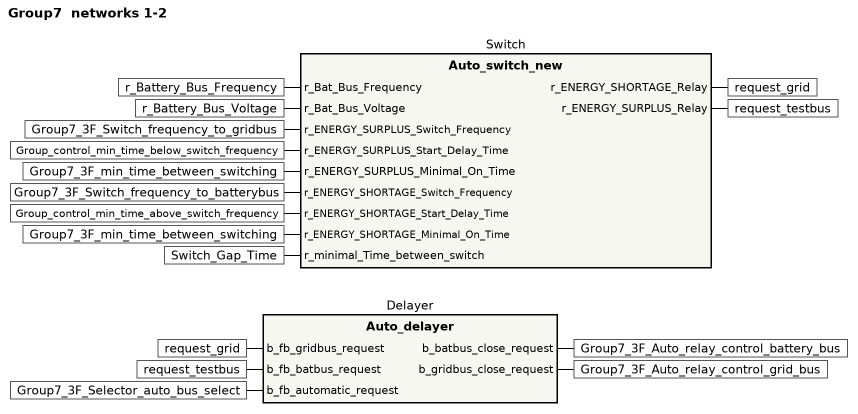
_FBD_ (* Function Block Diagram *)
NETWORK 1
	Switch:Auto_switch_new(r_Bat_Bus_Frequency: r_Battery_Bus_Frequency, r_Bat_Bus_Voltage: r_Battery_Bus_Voltage, r_ENERGY_SURPLUS_Switch_Frequency: Group7_3F_Switch_frequency_to_gridbus, r_ENERGY_SURPLUS_Start_Delay_Time: Group_control_min_time_below_switch_frequency, r_ENERGY_SURPLUS_Minimal_On_Time: Group7_3F_min_time_between_switching, r_ENERGY_SHORTAGE_Switch_Frequency: Group7_3F_Switch_frequency_to_batterybus, r_ENERGY_SHORTAGE_Start_Delay_Time: Group_control_min_time_above_switch_frequency, r_ENERGY_SHORTAGE_Minimal_On_Time: Group7_3F_min_time_between_switching, r_minimal_Time_between_switch: Switch_Gap_Time, r_ENERGY_SURPLUS_Relay => request_testbus) => request_grid
NETWORK 2
	Delayer:Auto_delayer(b_fb_gridbus_request: request_grid, b_fb_batbus_request: request_testbus, b_fb_automatic_request: Group7_3F_Selector_auto_bus_select, b_gridbus_close_request => Group7_3F_Auto_relay_control_grid_bus) => Group7_3F_Auto_relay_control_battery_bus
_END_FBD_
(* the same logic as Structured Text *)
(* Network 1 *)
Switch(r_Bat_Bus_Frequency := r_Battery_Bus_Frequency, r_Bat_Bus_Voltage := r_Battery_Bus_Voltage, r_ENERGY_SURPLUS_Switch_Frequency := Group7_3F_Switch_frequency_to_gridbus, r_ENERGY_SURPLUS_Start_Delay_Time := Group_control_min_time_below_switch_frequency, r_ENERGY_SURPLUS_Minimal_On_Time := Group7_3F_min_time_between_switching, r_ENERGY_SHORTAGE_Switch_Frequency := Group7_3F_Switch_frequency_to_batterybus, r_ENERGY_SHORTAGE_Start_Delay_Time := Group_control_min_time_above_switch_frequency, r_ENERGY_SHORTAGE_Minimal_On_Time := Group7_3F_min_time_between_switching, r_minimal_Time_between_switch := Switch_Gap_Time);
request_testbus := Switch.r_ENERGY_SURPLUS_Relay;
request_grid := Switch.r_ENERGY_SHORTAGE_Relay;
(* Network 2 *)
Delayer(b_fb_gridbus_request := request_grid, b_fb_batbus_request := request_testbus, b_fb_automatic_request := Group7_3F_Selector_auto_bus_select);
Group7_3F_Auto_relay_control_grid_bus := Delayer.b_gridbus_close_request;
Group7_3F_Auto_relay_control_battery_bus := Delayer.b_batbus_close_request;
END_PROGRAM

(* POU 04. Frequency based Bus Select/Group8, FBD *)
PROGRAM Group8
VAR

	request_grid: BOOL;
	request_testbus: BOOL;
	Delayer: Auto_delayer;
	Switch: Auto_switch_new;
END_VAR
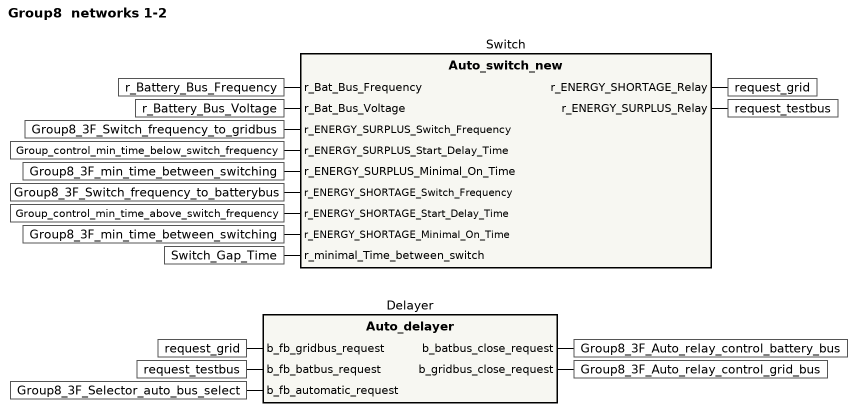
_FBD_ (* Function Block Diagram *)
NETWORK 1
	Switch:Auto_switch_new(r_Bat_Bus_Frequency: r_Battery_Bus_Frequency, r_Bat_Bus_Voltage: r_Battery_Bus_Voltage, r_ENERGY_SURPLUS_Switch_Frequency: Group8_3F_Switch_frequency_to_gridbus, r_ENERGY_SURPLUS_Start_Delay_Time: Group_control_min_time_below_switch_frequency, r_ENERGY_SURPLUS_Minimal_On_Time: Group8_3F_min_time_between_switching, r_ENERGY_SHORTAGE_Switch_Frequency: Group8_3F_Switch_frequency_to_batterybus, r_ENERGY_SHORTAGE_Start_Delay_Time: Group_control_min_time_above_switch_frequency, r_ENERGY_SHORTAGE_Minimal_On_Time: Group8_3F_min_time_between_switching, r_minimal_Time_between_switch: Switch_Gap_Time, r_ENERGY_SURPLUS_Relay => request_testbus) => request_grid
NETWORK 2
	Delayer:Auto_delayer(b_fb_gridbus_request: request_grid, b_fb_batbus_request: request_testbus, b_fb_automatic_request: Group8_3F_Selector_auto_bus_select, b_gridbus_close_request => Group8_3F_Auto_relay_control_grid_bus) => Group8_3F_Auto_relay_control_battery_bus
_END_FBD_
(* the same logic as Structured Text *)
(* Network 1 *)
Switch(r_Bat_Bus_Frequency := r_Battery_Bus_Frequency, r_Bat_Bus_Voltage := r_Battery_Bus_Voltage, r_ENERGY_SURPLUS_Switch_Frequency := Group8_3F_Switch_frequency_to_gridbus, r_ENERGY_SURPLUS_Start_Delay_Time := Group_control_min_time_below_switch_frequency, r_ENERGY_SURPLUS_Minimal_On_Time := Group8_3F_min_time_between_switching, r_ENERGY_SHORTAGE_Switch_Frequency := Group8_3F_Switch_frequency_to_batterybus, r_ENERGY_SHORTAGE_Start_Delay_Time := Group_control_min_time_above_switch_frequency, r_ENERGY_SHORTAGE_Minimal_On_Time := Group8_3F_min_time_between_switching, r_minimal_Time_between_switch := Switch_Gap_Time);
request_testbus := Switch.r_ENERGY_SURPLUS_Relay;
request_grid := Switch.r_ENERGY_SHORTAGE_Relay;
(* Network 2 *)
Delayer(b_fb_gridbus_request := request_grid, b_fb_batbus_request := request_testbus, b_fb_automatic_request := Group8_3F_Selector_auto_bus_select);
Group8_3F_Auto_relay_control_grid_bus := Delayer.b_gridbus_close_request;
Group8_3F_Auto_relay_control_battery_bus := Delayer.b_batbus_close_request;
END_PROGRAM

(* POU 04. Frequency based Bus Select/Group9, FBD *)
PROGRAM Group9
VAR

	request_grid: BOOL;
	request_testbus: BOOL;
	Delayer: Auto_delayer;
	Switch: Auto_switch_new;
END_VAR
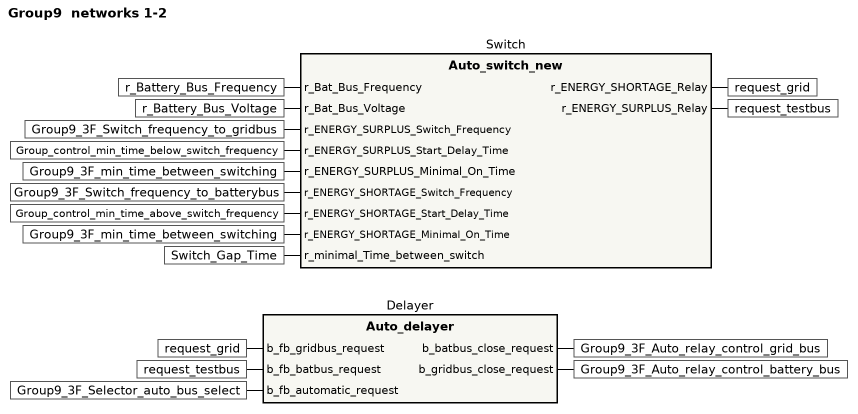
_FBD_ (* Function Block Diagram *)
NETWORK 1
	Switch:Auto_switch_new(r_Bat_Bus_Frequency: r_Battery_Bus_Frequency, r_Bat_Bus_Voltage: r_Battery_Bus_Voltage, r_ENERGY_SURPLUS_Switch_Frequency: Group9_3F_Switch_frequency_to_gridbus, r_ENERGY_SURPLUS_Start_Delay_Time: Group_control_min_time_below_switch_frequency, r_ENERGY_SURPLUS_Minimal_On_Time: Group9_3F_min_time_between_switching, r_ENERGY_SHORTAGE_Switch_Frequency: Group9_3F_Switch_frequency_to_batterybus, r_ENERGY_SHORTAGE_Start_Delay_Time: Group_control_min_time_above_switch_frequency, r_ENERGY_SHORTAGE_Minimal_On_Time: Group9_3F_min_time_between_switching, r_minimal_Time_between_switch: Switch_Gap_Time, r_ENERGY_SURPLUS_Relay => request_testbus) => request_grid
NETWORK 2
	Delayer:Auto_delayer(b_fb_gridbus_request: request_grid, b_fb_batbus_request: request_testbus, b_fb_automatic_request: Group9_3F_Selector_auto_bus_select, b_gridbus_close_request => Group9_3F_Auto_relay_control_battery_bus) => Group9_3F_Auto_relay_control_grid_bus
_END_FBD_
(* the same logic as Structured Text *)
(* Network 1 *)
Switch(r_Bat_Bus_Frequency := r_Battery_Bus_Frequency, r_Bat_Bus_Voltage := r_Battery_Bus_Voltage, r_ENERGY_SURPLUS_Switch_Frequency := Group9_3F_Switch_frequency_to_gridbus, r_ENERGY_SURPLUS_Start_Delay_Time := Group_control_min_time_below_switch_frequency, r_ENERGY_SURPLUS_Minimal_On_Time := Group9_3F_min_time_between_switching, r_ENERGY_SHORTAGE_Switch_Frequency := Group9_3F_Switch_frequency_to_batterybus, r_ENERGY_SHORTAGE_Start_Delay_Time := Group_control_min_time_above_switch_frequency, r_ENERGY_SHORTAGE_Minimal_On_Time := Group9_3F_min_time_between_switching, r_minimal_Time_between_switch := Switch_Gap_Time);
request_testbus := Switch.r_ENERGY_SURPLUS_Relay;
request_grid := Switch.r_ENERGY_SHORTAGE_Relay;
(* Network 2 *)
Delayer(b_fb_gridbus_request := request_grid, b_fb_batbus_request := request_testbus, b_fb_automatic_request := Group9_3F_Selector_auto_bus_select);
Group9_3F_Auto_relay_control_battery_bus := Delayer.b_gridbus_close_request;
Group9_3F_Auto_relay_control_grid_bus := Delayer.b_batbus_close_request;
END_PROGRAM

(* POU 07. Signal Lights/error_lights, ST *)
PROGRAM error_lights
VAR
END_VAR
	Control_panel_status_operational_led := 1;
	Control_panel_status_warning_led	:=0;
	Control_panel_status_error_led := 0;

IF r_Grid_Bus_Voltage < 220 THEN
		Control_panel_status_warning_led := 1;  (* Low Grid Voltage *)
END_IF

(* Should haves:
 Coupling LED flashing when sync command started (now implemented as warning light
*)

IF Bus_Connector_3F_Sync_close_requested <> Bus_Connector_3F_Sync_closed  THEN
	Control_panel_status_warning_led := 1;
END_IF

IF Group_control_Frequencybased_bus_selecting_state  THEN
(*--------------------------------------------------------------------------------------------------------------------------------------------------*)

IF Group1_3F_Selector_auto_bus_select THEN
	IF Group1_3F_Auto_relay_control_battery_bus <> Group1_3F_relay_state_battery_bus  THEN
			Control_panel_status_error_led := 1;
	END_IF

	IF Group1_3F_Auto_relay_control_grid_bus <> Group1_3F_relay_state_grid_bus  THEN
			Control_panel_status_error_led := 1;
	END_IF
END_IF



(*--------------------------------------------------------------------------------------------------------------------------------------------------*)
IF Group2_3F_Selector_auto_bus_select THEN
	IF Group2_3F_Auto_relay_control_battery_bus <> Group2_3F_relay_state_battery_bus  THEN
		Control_panel_status_error_led := 1;
	END_IF


	IF Group2_3F_Auto_relay_control_grid_bus <> Group2_3F_relay_state_grid_bus  THEN
		Control_panel_status_error_led := 1;
	END_IF
END_IF

(*--------------------------------------------------------------------------------------------------------------------------------------------------*)
IF Group3_3F_Selector_auto_bus_select THEN
	IF Group3_3F_Auto_relay_control_battery_bus <> Group3_3F_relay_state_battery_bus  THEN
		Control_panel_status_error_led := 1;
	END_IF

	IF Group3_3F_Auto_relay_control_grid_bus <> Group3_3F_relay_state_grid_bus  THEN
		Control_panel_status_error_led := 1;
	END_IF
END_IF



(*--------------------------------------------------------------------------------------------------------------------------------------------------*)
IF Group4_3F_Selector_auto_bus_select THEN
	IF Group4_3F_Auto_relay_control_battery_bus <> Group4_3F_relay_state_battery_bus  THEN
		Control_panel_status_error_led := 1;
	END_IF


	IF Group4_3F_Auto_relay_control_grid_bus <> Group4_3F_relay_state_grid_bus  THEN
		Control_panel_status_error_led := 1;
	END_IF
END_IF



(*--------------------------------------------------------------------------------------------------------------------------------------------------*)
IF Group5_3F_Selector_auto_bus_select THEN
	IF Group5_3F_Auto_relay_control_battery_bus <> Group5_3F_relay_state_battery_bus  THEN
		Control_panel_status_error_led := 1;
	END_IF


	IF Group5_3F_Auto_relay_control_grid_bus <> Group5_3F_relay_state_grid_bus  THEN
		Control_panel_status_error_led := 1;
	END_IF
END_IF



(*--------------------------------------------------------------------------------------------------------------------------------------------------*)
IF Group6_3F_Selector_auto_bus_select THEN
	IF Group6_3F_Auto_relay_control_battery_bus <> Group6_3F_relay_state_battery_bus  THEN
		Control_panel_status_error_led := 1;
	END_IF


	IF Group6_3F_Auto_relay_control_grid_bus <> Group6_3F_relay_state_grid_bus  THEN
		Control_panel_status_error_led := 1;
	END_IF
END_IF



(*--------------------------------------------------------------------------------------------------------------------------------------------------*)
IF Group7_3F_Selector_auto_bus_select THEN
	IF Group7_3F_Auto_relay_control_battery_bus <> Group7_3F_relay_state_battery_bus  THEN
		Control_panel_status_error_led := 1;
	END_IF


	IF Group7_3F_Auto_relay_control_grid_bus <> Group7_3F_relay_state_grid_bus  THEN
		Control_panel_status_error_led := 1;
	END_IF
END_IF



(*--------------------------------------------------------------------------------------------------------------------------------------------------*)
IF Group8_3F_Selector_auto_bus_select THEN
	IF Group8_3F_Auto_relay_control_battery_bus <> Group8_3F_relay_state_battery_bus  THEN
		Control_panel_status_error_led := 1;
	END_IF


	IF Group8_3F_Auto_relay_control_grid_bus <> Group8_3F_relay_state_grid_bus  THEN
		Control_panel_status_error_led := 1;
	END_IF
END_IF


(*--------------------------------------------------------------------------------------------------------------------------------------------------*)
IF Group9_3F_Selector_auto_bus_select THEN
	IF Group9_3F_Auto_relay_control_battery_bus <> Group9_3F_relay_state_battery_bus  THEN
		Control_panel_status_error_led := 1;
	END_IF


	IF Group9_3F_Auto_relay_control_grid_bus <> Group9_3F_relay_state_grid_bus  THEN
		Control_panel_status_error_led := 1;
	END_IF

END_IF

END_IF
END_PROGRAM

(* POU 01. PowerQualityMeasurements/run_PQ, ST *)
PROGRAM run_PQ
VAR
END_VAR
(* gridbus, batbus and connector monitoring *)
PQ_A();									(* postion : 11 *)
	r_Grid_Bus_Voltage					:= 	arMeasurementsGroupA[7];
	r_Grid_Bus_Frequency				:= 	arMeasurementsGroupA[13];

PQ_B();									(* postion : 1 *)
	r_Battery_Bus_Voltage				:= 	arMeasurementsGroupB[7];
	r_Battery_Bus_Frequency			:= 	arMeasurementsGroupB[13];

PQ_Janitza_Battery_Bus();

(* groups monitoring *)
PQ_1();									(* postion : 2 *)
PQ_2();									(* postion : 3 *)
PQ_3();									(* postion : 4 *)
PQ_4();									(* postion : 5 *)
PQ_5();									(* postion : 6 *)
PQ_6();									(* postion : 7 *)
PQ_7();									(* postion : 8 *)
PQ_8();									(* postion : 9 *)
PQ_9();									(* postion : 10 *)
END_PROGRAM

(* POU 01. PowerQualityMeasurements/PQ_A, FBD *)
PROGRAM PQ_A
VAR
	abProcessImageInput	AT %IW120		: ARRAY[0..23] OF BYTE;
	abProcessImageOutput 	AT %QW128		: ARRAY[0..23] OF BYTE;

	bToken										: BYTE;

	State_750_495 							: Fb_750_495_State;
		typ_750_495_State 						: typ_750_495_State;

	Configuration_750_495					: Fb_750_495_Configuration;
		typConfig_750_495						: typConfig_750_495;
		xReadyConfig								: BOOL;
		bFeedbackConfig							: BYTE;

	AC_Compact_01_750_495				: Fb_750_495_AC_Compact_01;
		rTotalActivePower							: REAL;
		rTotalReactivePower						: REAL;
		rTotalApparentPower						: REAL;
		rTotalPowerFactorPF						: REAL;
		rTotalActiveEnergy							: REAL;
		rTotalReactiveEnergy						: REAL;
		rTotalApparentEnergy						: REAL;
		rCurrentN									: REAL;
		xRotatingField								: BOOL;
		arCurrent									: ARRAY[1..3] OF REAL;
		axOvercurrent								: ARRAY[1..3] OF BOOL;
		arVoltage_L_N							: ARRAY[1..3] OF REAL;
		axUndervoltage							: ARRAY[1..3] OF BOOL;
		axOvervoltage								: ARRAY[1..3] OF BOOL;
		arActivePower								: ARRAY[1..3] OF REAL;
		arReactivePower							: ARRAY[1..3] OF REAL;
		arApparentPower							: ARRAY[1..3] OF REAL;
		arCosPhi									: ARRAY[1..3] OF REAL;
		arPowerFactorPF							: ARRAY[1..3] OF REAL;
		arFrequency								: ARRAY[1..3] OF REAL;
		axNoZero									: ARRAY[1..3] OF BOOL;
		axVoltSag									: ARRAY[1..3] OF BOOL;
		ai4Quadrant								: ARRAY[1..3] OF INT;

		xReadyCompact_01						: BOOL;
		abFeedbackCompact_01					: ARRAY[1..8] OF BYTE;


END_VAR
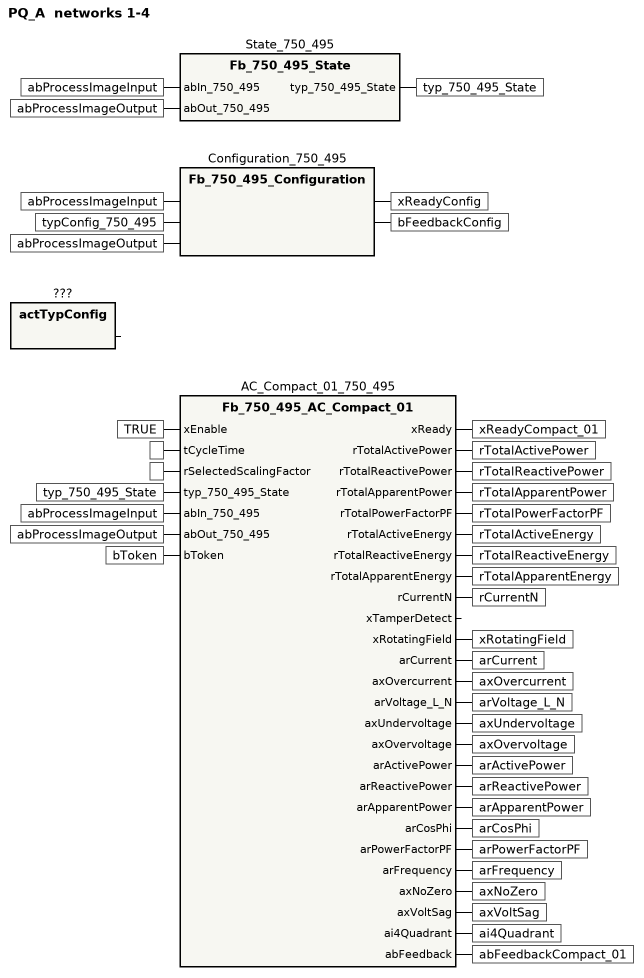
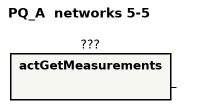
_FBD_ (* Function Block Diagram *)
NETWORK 1
	State_750_495:Fb_750_495_State(abIn_750_495: abProcessImageInput, abOut_750_495: abProcessImageOutput) => typ_750_495_State
NETWORK 2
	Configuration_750_495:Fb_750_495_Configuration(abProcessImageInput, typConfig_750_495, abProcessImageOutput, out 2 => bFeedbackConfig) => xReadyConfig
NETWORK 3
	???:actTypConfig()
NETWORK 4
	AC_Compact_01_750_495:Fb_750_495_AC_Compact_01(xEnable: TRUE, tCycleTime: , rSelectedScalingFactor: , typ_750_495_State: typ_750_495_State, abIn_750_495: abProcessImageInput, abOut_750_495: abProcessImageOutput, bToken: bToken, rTotalActivePower => rTotalActivePower, rTotalReactivePower => rTotalReactivePower, rTotalApparentPower => rTotalApparentPower, rTotalPowerFactorPF => rTotalPowerFactorPF, rTotalActiveEnergy => rTotalActiveEnergy, rTotalReactiveEnergy => rTotalReactiveEnergy, rTotalApparentEnergy => rTotalApparentEnergy, rCurrentN => rCurrentN, xRotatingField => xRotatingField, arCurrent => arCurrent, axOvercurrent => axOvercurrent, arVoltage_L_N => arVoltage_L_N, axUndervoltage => axUndervoltage, axOvervoltage => axOvervoltage, arActivePower => arActivePower, arReactivePower => arReactivePower, arApparentPower => arApparentPower, arCosPhi => arCosPhi, arPowerFactorPF => arPowerFactorPF, arFrequency => arFrequency, axNoZero => axNoZero, axVoltSag => axVoltSag, ai4Quadrant => ai4Quadrant, abFeedback => abFeedbackCompact_01) => xReadyCompact_01
NETWORK 5
	???:actGetMeasurements()
_END_FBD_
(* the same logic as Structured Text *)
(* Network 1 *)
State_750_495(abIn_750_495 := abProcessImageInput, abOut_750_495 := abProcessImageOutput);
typ_750_495_State := State_750_495.typ_750_495_State;
(* Network 2: see the listing above *)
(* Network 3: see the listing above *)
(* Network 4: see the listing above *)
(* Network 5: see the listing above *)
END_PROGRAM
ACTION actGetMeasurements:
arMeasurementsGroupA[1] := arActivePower[1];
arMeasurementsGroupA[2] := arActivePower[2];
arMeasurementsGroupA[3] := arActivePower[3];
arMeasurementsGroupA[4] := arReactivePower[1];
arMeasurementsGroupA[5] := arReactivePower[2];
arMeasurementsGroupA[6] := arReactivePower[3];
arMeasurementsGroupA[7] := arVoltage_L_N[1];
arMeasurementsGroupA[8] := arVoltage_L_N[2];
arMeasurementsGroupA[9] := arVoltage_L_N[3];
arMeasurementsGroupA[10] := arCurrent[1];
arMeasurementsGroupA[11] := arCurrent[2];
arMeasurementsGroupA[12] := arCurrent[3];
arMeasurementsGroupA[13] := arFrequency[1];
arMeasurementsGroupA[14] := arFrequency[2];
arMeasurementsGroupA[15] := arFrequency[3];
arMeasurementsGroupA[16] := rTotalActiveEnergy;
arMeasurementsGroupA[17] := BOOL_TO_REAL(xRotatingField);
arMeasurementsGroupA[18] := rTotalReactiveEnergy;
END_ACTION
ACTION actTypConfig:
typConfig_750_495.typChannelConfig[1].xEnableUserScaling:= TRUE;
typConfig_750_495.typChannelConfig[1].wCurrentTransformerRatio :=CurrentRatioPQA;

typConfig_750_495.typChannelConfig[2].xEnableUserScaling:= TRUE;
typConfig_750_495.typChannelConfig[2].wCurrentTransformerRatio :=CurrentRatioPQA;

typConfig_750_495.typChannelConfig[3].xEnableUserScaling:= TRUE;
typConfig_750_495.typChannelConfig[3].wCurrentTransformerRatio :=CurrentRatioPQA;

typConfig_750_495.xWriteConfig := TRUE;
END_ACTION

(* POU 01. PowerQualityMeasurements/PQ_B, FBD *)
PROGRAM PQ_B
VAR
	abProcessImageInput	AT %IW0			: ARRAY[0..23] OF BYTE;
	abProcessImageOutput 	AT %QW8 			: ARRAY[0..23] OF BYTE;

	bToken										: BYTE;

	State_750_495 							: Fb_750_495_State;
		typ_750_495_State 						: typ_750_495_State;

	Configuration_750_495					: Fb_750_495_Configuration;
		typConfig_750_495						: typConfig_750_495;
		xReadyConfig								: BOOL;
		bFeedbackConfig							: BYTE;

	AC_Compact_01_750_495				: Fb_750_495_AC_Compact_01;
		rTotalActivePower							: REAL;
		rTotalReactivePower						: REAL;
		rTotalApparentPower						: REAL;
		rTotalPowerFactorPF						: REAL;
		rTotalActiveEnergy							: REAL;
		rTotalReactiveEnergy						: REAL;
		rTotalApparentEnergy						: REAL;
		rCurrentN									: REAL;
		xRotatingField								: BOOL;
		arCurrent									: ARRAY[1..3] OF REAL;
		axOvercurrent								: ARRAY[1..3] OF BOOL;
		arVoltage_L_N							: ARRAY[1..3] OF REAL;
		axUndervoltage							: ARRAY[1..3] OF BOOL;
		axOvervoltage								: ARRAY[1..3] OF BOOL;
		arActivePower								: ARRAY[1..3] OF REAL;
		arReactivePower							: ARRAY[1..3] OF REAL;
		arApparentPower							: ARRAY[1..3] OF REAL;
		arCosPhi									: ARRAY[1..3] OF REAL;
		arPowerFactorPF							: ARRAY[1..3] OF REAL;
		arFrequency								: ARRAY[1..3] OF REAL;
		axNoZero									: ARRAY[1..3] OF BOOL;
		axVoltSag									: ARRAY[1..3] OF BOOL;
		ai4Quadrant								: ARRAY[1..3] OF INT;

		xReadyCompact_01						: BOOL;
		abFeedbackCompact_01					: ARRAY[1..8] OF BYTE;


END_VAR
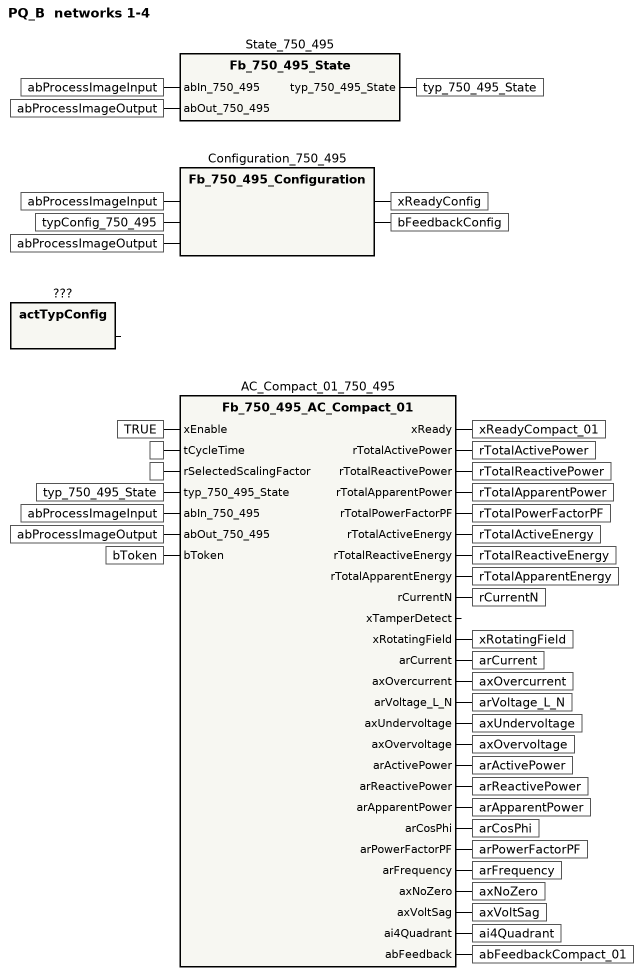
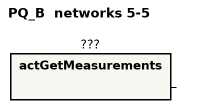
_FBD_ (* Function Block Diagram *)
NETWORK 1
	State_750_495:Fb_750_495_State(abIn_750_495: abProcessImageInput, abOut_750_495: abProcessImageOutput) => typ_750_495_State
NETWORK 2
	Configuration_750_495:Fb_750_495_Configuration(abProcessImageInput, typConfig_750_495, abProcessImageOutput, out 2 => bFeedbackConfig) => xReadyConfig
NETWORK 3
	???:actTypConfig()
NETWORK 4
	AC_Compact_01_750_495:Fb_750_495_AC_Compact_01(xEnable: TRUE, tCycleTime: , rSelectedScalingFactor: , typ_750_495_State: typ_750_495_State, abIn_750_495: abProcessImageInput, abOut_750_495: abProcessImageOutput, bToken: bToken, rTotalActivePower => rTotalActivePower, rTotalReactivePower => rTotalReactivePower, rTotalApparentPower => rTotalApparentPower, rTotalPowerFactorPF => rTotalPowerFactorPF, rTotalActiveEnergy => rTotalActiveEnergy, rTotalReactiveEnergy => rTotalReactiveEnergy, rTotalApparentEnergy => rTotalApparentEnergy, rCurrentN => rCurrentN, xRotatingField => xRotatingField, arCurrent => arCurrent, axOvercurrent => axOvercurrent, arVoltage_L_N => arVoltage_L_N, axUndervoltage => axUndervoltage, axOvervoltage => axOvervoltage, arActivePower => arActivePower, arReactivePower => arReactivePower, arApparentPower => arApparentPower, arCosPhi => arCosPhi, arPowerFactorPF => arPowerFactorPF, arFrequency => arFrequency, axNoZero => axNoZero, axVoltSag => axVoltSag, ai4Quadrant => ai4Quadrant, abFeedback => abFeedbackCompact_01) => xReadyCompact_01
NETWORK 5
	???:actGetMeasurements()
_END_FBD_
(* the same logic as Structured Text *)
(* Network 1 *)
State_750_495(abIn_750_495 := abProcessImageInput, abOut_750_495 := abProcessImageOutput);
typ_750_495_State := State_750_495.typ_750_495_State;
(* Network 2: see the listing above *)
(* Network 3: see the listing above *)
(* Network 4: see the listing above *)
(* Network 5: see the listing above *)
END_PROGRAM
ACTION actGetMeasurements:
arMeasurementsGroupB[1] := arActivePower[1];
arMeasurementsGroupB[2] := arActivePower[2];
arMeasurementsGroupB[3] := arActivePower[3];
arMeasurementsGroupB[4] := arReactivePower[1];
arMeasurementsGroupB[5] := arReactivePower[2];
arMeasurementsGroupB[6] := arReactivePower[3];
arMeasurementsGroupB[7] := arVoltage_L_N[1];
arMeasurementsGroupB[8] := arVoltage_L_N[2];
arMeasurementsGroupB[9] := arVoltage_L_N[3];
arMeasurementsGroupB[10] := arCurrent[1];
arMeasurementsGroupB[11] := arCurrent[2];
arMeasurementsGroupB[12] := arCurrent[3];
arMeasurementsGroupB[13] := arFrequency[1];
arMeasurementsGroupB[14] := arFrequency[2];
arMeasurementsGroupB[15] := arFrequency[3];
arMeasurementsGroupB[16] := rTotalActiveEnergy;
arMeasurementsGroupB[17] := BOOL_TO_REAL(xRotatingField);
arMeasurementsGroupB[18] := rTotalReactiveEnergy;
END_ACTION
ACTION actTypConfig:
typConfig_750_495.typChannelConfig[1].xEnableUserScaling:= TRUE;
typConfig_750_495.typChannelConfig[1].wCurrentTransformerRatio :=CurrentRatioPQB;

typConfig_750_495.typChannelConfig[2].xEnableUserScaling:= TRUE;
typConfig_750_495.typChannelConfig[2].wCurrentTransformerRatio :=CurrentRatioPQB;

typConfig_750_495.typChannelConfig[3].xEnableUserScaling:= TRUE;
typConfig_750_495.typChannelConfig[3].wCurrentTransformerRatio :=CurrentRatioPQB;

typConfig_750_495.xWriteConfig := TRUE;
END_ACTION

(* POU 01. PowerQualityMeasurements/PQ_Janitza_Battery_Bus, ST *)
PROGRAM PQ_Janitza_Battery_Bus
(*  Link to modbus example: https://wiki.janitza.de/display/GRIDVIS70EN/UMG+604+-+Modbus  *)
(* Link to modbus commands/registers:  https://www.janitza.com/manuals.html          UMG 509 Modbus address and formulary (English)  *)
VAR

END_VAR
(* to be implemented: arMeasurementsJanitza[x] := Janitza_Modbus[y];*)


(* to be matched from janitza modbus  <<  see janitza modbus object*)

Bus_Connector_L1_P := -1 * MBCFG_Janitza_UMG5090.PactiveL1;
Bus_Connector_L2_P := -1 * MBCFG_Janitza_UMG5090.PactiveL2;
Bus_Connector_L3_P := -1 * MBCFG_Janitza_UMG5090.PactiveL3;
Bus_Connector_L1_Q := -1 * MBCFG_Janitza_UMG5090.PreactiveL1;
Bus_Connector_L2_Q :=-1 * MBCFG_Janitza_UMG5090.PreactiveL2;
Bus_Connector_L3_Q :=-1 * MBCFG_Janitza_UMG5090.PreactiveL3;
Bus_Connector_L1_V := MBCFG_Janitza_UMG5090.VoltageL1;
Bus_Connector_L2_V := MBCFG_Janitza_UMG5090.VoltageL2;
Bus_Connector_L3_V := MBCFG_Janitza_UMG5090.VoltageL3;
Bus_Connector_L1_I := MBCFG_Janitza_UMG5090.PhaseCurrentL1;
Bus_Connector_L2_I := MBCFG_Janitza_UMG5090.PhaseCurrentL2;
Bus_Connector_L3_I := MBCFG_Janitza_UMG5090.PhaseCurrentL3;
Bus_Connector_L1_f :=MBCFG_Janitza_UMG5090.Frequency;
Bus_Connector_L2_f :=MBCFG_Janitza_UMG5090.Frequency;
Bus_Connector_L3_f :=MBCFG_Janitza_UMG5090.Frequency;
Bus_Connector_3F_Field_Rotation :=MBCFG_Janitza_UMG5090.FieldRotation;
Bus_Connector_3F_CosPhi :=MBCFG_Janitza_UMG5090.CosPihL1;
(*
Can be implemented when required:

Bus_Connector_L3_f :=MBCFG_Janitza_UMG5090.CosPihL2;
Bus_Connector_L3_f :=MBCFG_Janitza_UMG5090.CosPihL3;
Bus_Connector_L3_f :=MBCFG_Janitza_UMG5090.Frequency;
Bus_Connector_L3_f :=MBCFG_Janitza_UMG5090.PactivetTot;
Bus_Connector_L3_f :=MBCFG_Janitza_UMG5090.PactivetTotL4;

*)
END_PROGRAM

(* POU Generated Code/Ethernet/MBCFG_Janitza_UMG5090, ST *)
PROGRAM MBCFG_Janitza_UMG5090(* generated by config one prg for each slave *)

VAR_INPUT

END_VAR

VAR_OUTPUT
       PactiveL1       :    REAL;       (**) 
       PactiveL2       :    REAL;       (**) 
       PactiveL3       :    REAL;       (**) 
       PreactiveL1       :    REAL;       (**) 
       PreactiveL2       :    REAL;       (**) 
       PreactiveL3       :    REAL;       (**) 
       VoltageL1       :    REAL;       (**) 
       VoltageL2       :    REAL;       (**) 
       VoltageL3       :    REAL;       (**) 
       VoltageL4       :    REAL;       (**) 
       PhaseCurrentL1       :    REAL;       (**) 
       PhaseCurrentL2       :    REAL;       (**) 
       PhaseCurrentL3       :    REAL;       (**) 
       PhaseCurrentLN       :    REAL;       (**) 
       FieldRotation       :    REAL;       (**)
       CosPihL1       :    REAL;       (**) 
       CosPihL2       :    REAL;       (**) 
       CosPihL3       :    REAL;       (**) 
       Frequency       :    REAL;       (**) 
       PactivetTot       :    REAL;       (**) 
       PactivetTotL4       :    REAL;       (**) 

